IF NOT Execute THEN
	eState := STATE_RESETTING;
ELSIF _Error THEN
	eState := STATE_ERROR;
ELSIF _Abort THEN
	eState := STATE_ABORTING;
ELSIF _Executed THEN
	eState := STATE_DONE;
END_IF
END_METHOD

METHOD  M_STATE_RESETTING
VAR_INPUT
END_VAR
Busy := FALSE;
Aborted := FALSE;
Error := FALSE;

CASE uiResettingStep OF
	0:
		ModeRequestValid := FALSE;
		TON_WaitModeSwitch.IN := FALSE;

		uiResettingStep := 100;

	100:
		_ResetCompleted := TRUE;
END_CASE

IF _ResetCompleted THEN
	eState := STATE_DORMANT;
END_IF
END_METHOD

END_FUNCTION_BLOCK

// ---- Library/30_Simulation/10_IOSim/FB_SimulatedIO.TcPOU
(*
    FB_SimulatedIO — 數位孿生 IO 模擬層
    =====================================================
    每個 PLC 週期：
      1. 將所有安全門、氣壓 Input bit 強制為 TRUE（使機器可啟動）
      2. 監看 GVL_Output.uniDO.stDO 的 Valve 輸出位元
      3. 透過 TON 延遲後，回寫對應的 GVL_Input.uniDI.stDI 感測器位元
    使用方式：在 FB_MachineControl 主體中：
      IF EnableSimulation THEN fbSimulatedIO(); END_IF
*)
FUNCTION_BLOCK FB_SimulatedIO
VAR_INPUT
END_VAR
VAR_OUTPUT
END_VAR
VAR
    // ----- 安全輸入注入用旗標 -----
    _tSafetyInject : TON; // 短延遲確保每次都會執行注入

    // ----- Group 1: Double valve, FrontSensor + RearSensor -----
    // fbUpCV_DiameterHoriz
    tonDiamHoriz_Ext : TON;
    tonDiamHoriz_Ret : TON;
    // fbTransmitCV_CamaraHoriz
    tonCamaraHoriz_Ext : TON;
    tonCamaraHoriz_Ret : TON;

    // ----- Group 2: Single valve, FrontSensor + RearSensor -----
    // fbUpCV_DiameterVert
    tonDiamVert_Ext : TON;
    tonDiamVert_Ret : TON;
    // fbStackPush
    tonStackPush_Ext : TON;
    tonStackPush_Ret : TON;
    // fbAllocateRobot_LeftVert1
    tonLV1_Ext : TON;
    tonLV1_Ret : TON;
    // fbAllocateRobot_LeftVert2
    tonLV2_Ext : TON;
    tonLV2_Ret : TON;
    // fbAllocateRobot_RightVert1
    tonRV1_Ext : TON;
    tonRV1_Ret : TON;
    // fbAllocateRobot_RightVert2
    tonRV2_Ext : TON;
    tonRV2_Ret : TON;
    // fbRoundBelt_WorkZone_Plug
    tonWZPlug_Ext : TON;
    tonWZPlug_Ret : TON;
    // fbRoundBelt_ChargeZone_Plug
    tonCZPlug_Ext : TON;
    tonCZPlug_Ret : TON;
    // fbRoundBelt_TransmitCVZone_Plug
    tonTCVPlug_Ext : TON;
    tonTCVPlug_Ret : TON;
    // fbOutRobot_AsideVert
    tonAsideVert_Ext : TON;
    tonAsideVert_Ret : TON;
    // fbOutRobot_BsideVert
    tonBsideVert_Ext : TON;
    tonBsideVert_Ret : TON;

    // ----- Group 3: Double valve, RearSensor only -----
    // fbUpCV_Block1/2/3
    tonUpBlock1_Ext : TON;
    tonUpBlock1_Ret : TON;
    tonUpBlock2_Ext : TON;
    tonUpBlock2_Ret : TON;
    tonUpBlock3_Ext : TON;
    tonUpBlock3_Ret : TON;
    // fbLowCV_Block1/2
    tonLowBlock1_Ext : TON;
    tonLowBlock1_Ret : TON;
    tonLowBlock2_Ext : TON;
    tonLowBlock2_Ret : TON;
    // fbOutRobot_AsideClamp / BsideClamp
    tonAsideClamp_Ext : TON;
    tonAsideClamp_Ret : TON;
    tonBsideClamp_Ext : TON;
    tonBsideClamp_Ret : TON;

    // ----- Group 4: Single valve, RearSensor only -----
    // fbPullOutCV_AsideBlock / BsideBlock
    tonPullAside_Ext : TON;
    tonPullAside_Ret : TON;
    tonPullBside_Ext : TON;
    tonPullBside_Ret : TON;
    // fbRoundBelt_WorkZone_Press
    tonWZPress_Ext : TON;
    tonWZPress_Ret : TON;
    // fbDifferentSizeCV_Block1
    tonDiffBlock1_Ext : TON;
    tonDiffBlock1_Ret : TON;
    // fbSameSizeCV_Block1 / Block2
    tonSameBlock1_Ext : TON;
    tonSameBlock1_Ret : TON;
    tonSameBlock2_Ext : TON;
    tonSameBlock2_Ret : TON;
    // fbTurntable_Press
    tonTTPress_Ext : TON;
    tonTTPress_Ret : TON;
END_VAR
VAR CONSTANT
    tCYL_DELAY : TIME := T#300MS; // 汽缸模擬動作延遲（可依需求調整）
END_VAR

// ═══════════════════════════════════════════════════════════════
// 1. 安全輸入每週期強制 TRUE — 讓機器可以在無硬體下啟動
// ═══════════════════════════════════════════════════════════════
GVL_Input.uniDI.stDI.bSafetyDoor1  := TRUE;
GVL_Input.uniDI.stDI.bSafetyDoor2  := TRUE;
GVL_Input.uniDI.stDI.bSafetyDoor3  := TRUE;
GVL_Input.uniDI.stDI.bSafetyDoor4  := TRUE;
GVL_Input.uniDI.stDI.bSafetyDoor5  := TRUE;
GVL_Input.uniDI.stDI.bSafetyDoor6  := TRUE;
GVL_Input.uniDI.stDI.bSafetyDoor7  := TRUE;
GVL_Input.uniDI.stDI.bSafetyDoor8  := TRUE;
GVL_Input.uniDI.stDI.bSafetyDoor9  := TRUE;
GVL_Input.uniDI.stDI.bSafetyDoor10 := TRUE;
GVL_Input.uniDI.stDI.bSafetyDoor11 := TRUE;
GVL_Input.uniDI.stDI.bSafetyDoor12 := TRUE;
GVL_Input.uniDI.stDI.bSafetyDoor13 := TRUE;
GVL_Input.uniDI.stDI.bSafetyDoor14 := TRUE;
GVL_Input.uniDI.stDI.bAllocate_Electrical_Cabinet_SafetyDoor      := TRUE;
GVL_Input.uniDI.stDI.bShippingRobot_ElectricalCabinet_SafetyDoor  := TRUE;
GVL_Input.uniDI.stDI.bStorage_AirPressure_Ready   := TRUE;
GVL_Input.uniDI.stDI.bAllocate_AirPressure_Ready  := TRUE;

// ═══════════════════════════════════════════════════════════════
// 2. 汽缸 IO 模擬  (讀 Output Valve → 延遲 → 寫 Input Sensor)
//    每個 TON:  _Ext 監看伸出命令, _Ret 監看縮回命令
// ═══════════════════════════════════════════════════════════════

// ─── Group 1: Double valve, FrontSensor + RearSensor ─────────

// fbUpCV_DiameterHoriz (雙閥, 兩端感測器)
tonDiamHoriz_Ext(IN := GVL_Output.uniDO.stDO.bUpCV_DiameterHoriz_Extend_Valve, PT := tCYL_DELAY);
tonDiamHoriz_Ret(IN := GVL_Output.uniDO.stDO.bUpCV_DiameterHoriz_Retract_Valve, PT := tCYL_DELAY);
IF tonDiamHoriz_Ext.Q THEN
    GVL_Input.uniDI.stDI.bUpCV_DiameterHoriz_FrontSensor := TRUE;
    GVL_Input.uniDI.stDI.bUpCV_DiameterHoriz_RearSensor  := FALSE;
ELSIF tonDiamHoriz_Ret.Q THEN
    GVL_Input.uniDI.stDI.bUpCV_DiameterHoriz_FrontSensor := FALSE;
    GVL_Input.uniDI.stDI.bUpCV_DiameterHoriz_RearSensor  := TRUE;
END_IF

// fbTransmitCV_CamaraHoriz (雙閥, 兩端感測器)
tonCamaraHoriz_Ext(IN := GVL_Output.uniDO.stDO.bTransmitCV_CamaraHorizDifferentSide_Valve, PT := tCYL_DELAY);
tonCamaraHoriz_Ret(IN := GVL_Output.uniDO.stDO.bTransmitCV_CamaraHorizSameSizeSide_Valve,  PT := tCYL_DELAY);
IF tonCamaraHoriz_Ext.Q THEN
    GVL_Input.uniDI.stDI.bTransmit_CamaraHorizDifferentSizeSide_Sensor := TRUE;
    GVL_Input.uniDI.stDI.bTransmit_CamaraHorizSameSizeSide_Sensor      := FALSE;
ELSIF tonCamaraHoriz_Ret.Q THEN
    GVL_Input.uniDI.stDI.bTransmit_CamaraHorizDifferentSizeSide_Sensor := FALSE;
    GVL_Input.uniDI.stDI.bTransmit_CamaraHorizSameSizeSide_Sensor      := TRUE;
END_IF

// ─── Group 2: Single valve, FrontSensor + RearSensor ─────────

// fbUpCV_DiameterVert
tonDiamVert_Ext(IN :=      GVL_Output.uniDO.stDO.bUpCV_DiameterVert_Valve, PT := tCYL_DELAY);
tonDiamVert_Ret(IN := NOT  GVL_Output.uniDO.stDO.bUpCV_DiameterVert_Valve, PT := tCYL_DELAY);
IF tonDiamVert_Ext.Q THEN
    GVL_Input.uniDI.stDI.bUpCV_DiameterVert_FrontSensor := TRUE;
    GVL_Input.uniDI.stDI.bUpCV_DiameterVert_RearSensor  := FALSE;
ELSIF tonDiamVert_Ret.Q THEN
    GVL_Input.uniDI.stDI.bUpCV_DiameterVert_FrontSensor := FALSE;
    GVL_Input.uniDI.stDI.bUpCV_DiameterVert_RearSensor  := TRUE;
END_IF

// fbStackPush
tonStackPush_Ext(IN :=      GVL_Output.uniDO.stDO.bStackPush_Valve, PT := tCYL_DELAY);
tonStackPush_Ret(IN := NOT  GVL_Output.uniDO.stDO.bStackPush_Valve, PT := tCYL_DELAY);
IF tonStackPush_Ext.Q THEN
    GVL_Input.uniDI.stDI.bStackPush_Pusher_FrontSensor := TRUE;
    GVL_Input.uniDI.stDI.bStackPush_Pusher_RearSensor  := FALSE;
ELSIF tonStackPush_Ret.Q THEN
    GVL_Input.uniDI.stDI.bStackPush_Pusher_FrontSensor := FALSE;
    GVL_Input.uniDI.stDI.bStackPush_Pusher_RearSensor  := TRUE;
END_IF

// fbAllocateRobot_LeftVert1
tonLV1_Ext(IN :=      GVL_Output.uniDO.stDO.bAllocateRobot_LeftVert1_Valve, PT := tCYL_DELAY);
tonLV1_Ret(IN := NOT  GVL_Output.uniDO.stDO.bAllocateRobot_LeftVert1_Valve, PT := tCYL_DELAY);
IF tonLV1_Ext.Q THEN
    GVL_Input.uniDI.stDI.bAllocateRobot_LeftVert1_LowSensor  := TRUE;
    GVL_Input.uniDI.stDI.bAllocateRobot_LeftVert1_HighSensor := FALSE;
ELSIF tonLV1_Ret.Q THEN
    GVL_Input.uniDI.stDI.bAllocateRobot_LeftVert1_LowSensor  := FALSE;
    GVL_Input.uniDI.stDI.bAllocateRobot_LeftVert1_HighSensor := TRUE;
END_IF

// fbAllocateRobot_LeftVert2
tonLV2_Ext(IN :=      GVL_Output.uniDO.stDO.bAllocateRobot_LeftVert2_Valve, PT := tCYL_DELAY);
tonLV2_Ret(IN := NOT  GVL_Output.uniDO.stDO.bAllocateRobot_LeftVert2_Valve, PT := tCYL_DELAY);
IF tonLV2_Ext.Q THEN
    GVL_Input.uniDI.stDI.bAllocateRobot_LeftVert2_LowSensor  := TRUE;
    GVL_Input.uniDI.stDI.bAllocateRobot_LeftVert2_HighSensor := FALSE;
ELSIF tonLV2_Ret.Q THEN
    GVL_Input.uniDI.stDI.bAllocateRobot_LeftVert2_LowSensor  := FALSE;
    GVL_Input.uniDI.stDI.bAllocateRobot_LeftVert2_HighSensor := TRUE;
END_IF

// fbAllocateRobot_RightVert1
tonRV1_Ext(IN :=      GVL_Output.uniDO.stDO.bAllocateRobot_RightVert1_Valve, PT := tCYL_DELAY);
tonRV1_Ret(IN := NOT  GVL_Output.uniDO.stDO.bAllocateRobot_RightVert1_Valve, PT := tCYL_DELAY);
IF tonRV1_Ext.Q THEN
    GVL_Input.uniDI.stDI.bAllocateRobot_RightVert1_LowSensor  := TRUE;
    GVL_Input.uniDI.stDI.bAllocateRobot_RightVert1_HighSensor := FALSE;
ELSIF tonRV1_Ret.Q THEN
    GVL_Input.uniDI.stDI.bAllocateRobot_RightVert1_LowSensor  := FALSE;
    GVL_Input.uniDI.stDI.bAllocateRobot_RightVert1_HighSensor := TRUE;
END_IF

// fbAllocateRobot_RightVert2
tonRV2_Ext(IN :=      GVL_Output.uniDO.stDO.bAllocateRobot_RightVert2_Valve, PT := tCYL_DELAY);
tonRV2_Ret(IN := NOT  GVL_Output.uniDO.stDO.bAllocateRobot_RightVert2_Valve, PT := tCYL_DELAY);
IF tonRV2_Ext.Q THEN
    GVL_Input.uniDI.stDI.bAllocateRobot_RightVert2_LowSensor  := TRUE;
    GVL_Input.uniDI.stDI.bAllocateRobot_RightVert2_HighSensor := FALSE;
ELSIF tonRV2_Ret.Q THEN
    GVL_Input.uniDI.stDI.bAllocateRobot_RightVert2_LowSensor  := FALSE;
    GVL_Input.uniDI.stDI.bAllocateRobot_RightVert2_HighSensor := TRUE;
END_IF

// fbRoundBelt_WorkZone_Plug
tonWZPlug_Ext(IN :=      GVL_Output.uniDO.stDO.bRoundBelt_WorkZone_Plug_Valve, PT := tCYL_DELAY);
tonWZPlug_Ret(IN := NOT  GVL_Output.uniDO.stDO.bRoundBelt_WorkZone_Plug_Valve, PT := tCYL_DELAY);
IF tonWZPlug_Ext.Q THEN
    GVL_Input.uniDI.stDI.bRoundBelt_WorkZonePlug_frontSensor := TRUE;
    GVL_Input.uniDI.stDI.bRoundBelt_WorkZonePlug_RearSensor  := FALSE;
ELSIF tonWZPlug_Ret.Q THEN
    GVL_Input.uniDI.stDI.bRoundBelt_WorkZonePlug_frontSensor := FALSE;
    GVL_Input.uniDI.stDI.bRoundBelt_WorkZonePlug_RearSensor  := TRUE;
END_IF

// fbRoundBelt_ChargeZone_Plug
tonCZPlug_Ext(IN :=      GVL_Output.uniDO.stDO.bRoundBelt_ChargeZone_Plug_Valve, PT := tCYL_DELAY);
tonCZPlug_Ret(IN := NOT  GVL_Output.uniDO.stDO.bRoundBelt_ChargeZone_Plug_Valve, PT := tCYL_DELAY);
IF tonCZPlug_Ext.Q THEN
    GVL_Input.uniDI.stDI.bRoundBelt_ChangeZonePlug_FrontSensor := TRUE;
    GVL_Input.uniDI.stDI.bRoundBelt_ChangeZonePlug_RearSensor  := FALSE;
ELSIF tonCZPlug_Ret.Q THEN
    GVL_Input.uniDI.stDI.bRoundBelt_ChangeZonePlug_FrontSensor := FALSE;
    GVL_Input.uniDI.stDI.bRoundBelt_ChangeZonePlug_RearSensor  := TRUE;
END_IF

// fbRoundBelt_TransmitCVZone_Plug
tonTCVPlug_Ext(IN :=      GVL_Output.uniDO.stDO.bRoundBelt_TransmitCVZone_Plug_Valve, PT := tCYL_DELAY);
tonTCVPlug_Ret(IN := NOT  GVL_Output.uniDO.stDO.bRoundBelt_TransmitCVZone_Plug_Valve, PT := tCYL_DELAY);
IF tonTCVPlug_Ext.Q THEN
    GVL_Input.uniDI.stDI.bRoundBelt_TransmitCVZonePlug_FrontSensor := TRUE;
    GVL_Input.uniDI.stDI.bRoundBelt_TransmitCVZonePlug_RearSensor  := FALSE;
ELSIF tonTCVPlug_Ret.Q THEN
    GVL_Input.uniDI.stDI.bRoundBelt_TransmitCVZonePlug_FrontSensor := FALSE;
    GVL_Input.uniDI.stDI.bRoundBelt_TransmitCVZonePlug_RearSensor  := TRUE;
END_IF

// fbOutRobot_AsideVert (FrontSensor=Low, RearSensor=High)
tonAsideVert_Ext(IN :=      GVL_Output.uniDO.stDO.bOutRobot_AsideVert_Valve, PT := tCYL_DELAY);
tonAsideVert_Ret(IN := NOT  GVL_Output.uniDO.stDO.bOutRobot_AsideVert_Valve, PT := tCYL_DELAY);
IF tonAsideVert_Ext.Q THEN
    GVL_Input.uniDI.stDI.bOutRobot_AsideVert_LowSensor  := TRUE;
    GVL_Input.uniDI.stDI.bOutRobot_AsideVert_HighSensor := FALSE;
ELSIF tonAsideVert_Ret.Q THEN
    GVL_Input.uniDI.stDI.bOutRobot_AsideVert_LowSensor  := FALSE;
    GVL_Input.uniDI.stDI.bOutRobot_AsideVert_HighSensor := TRUE;
END_IF

// fbOutRobot_BsideVert (FrontSensor=Low, RearSensor=High)
tonBsideVert_Ext(IN :=      GVL_Output.uniDO.stDO.bOutRobot_BsideVert_Valve, PT := tCYL_DELAY);
tonBsideVert_Ret(IN := NOT  GVL_Output.uniDO.stDO.bOutRobot_BsideVert_Valve, PT := tCYL_DELAY);
IF tonBsideVert_Ext.Q THEN
    GVL_Input.uniDI.stDI.bOutRobot_BsideVert_LowSensor  := TRUE;
    GVL_Input.uniDI.stDI.bOutRobot_BsideVert_HighSensor := FALSE;
ELSIF tonBsideVert_Ret.Q THEN
    GVL_Input.uniDI.stDI.bOutRobot_BsideVert_LowSensor  := FALSE;
    GVL_Input.uniDI.stDI.bOutRobot_BsideVert_HighSensor := TRUE;
END_IF

// ─── Group 3: Double valve, RearSensor only ───────────────────

// fbUpCV_Block1  (Up=Extend=front, Down=Retract=rear)
tonUpBlock1_Ext(IN := GVL_Output.uniDO.stDO.bUpCV_Block1_Up_Valve,   PT := tCYL_DELAY);
tonUpBlock1_Ret(IN := GVL_Output.uniDO.stDO.bUpCV_Block1_Down_Valve, PT := tCYL_DELAY);
IF tonUpBlock1_Ext.Q THEN
    GVL_Input.uniDI.stDI.bUpCV_Block1_RearSensor := FALSE;
ELSIF tonUpBlock1_Ret.Q THEN
    GVL_Input.uniDI.stDI.bUpCV_Block1_RearSensor := TRUE;
END_IF

// fbUpCV_Block2
tonUpBlock2_Ext(IN := GVL_Output.uniDO.stDO.bUpCV_Block2_Up_Valve,   PT := tCYL_DELAY);
tonUpBlock2_Ret(IN := GVL_Output.uniDO.stDO.bUpCV_Block2_Down_Valve, PT := tCYL_DELAY);
IF tonUpBlock2_Ext.Q THEN
    GVL_Input.uniDI.stDI.bUpCV_Block2_RearSensor := FALSE;
ELSIF tonUpBlock2_Ret.Q THEN
    GVL_Input.uniDI.stDI.bUpCV_Block2_RearSensor := TRUE;
END_IF

// fbUpCV_Block3
tonUpBlock3_Ext(IN := GVL_Output.uniDO.stDO.bUpCV_Block3_Up_Valve,   PT := tCYL_DELAY);
tonUpBlock3_Ret(IN := GVL_Output.uniDO.stDO.bUpCV_Block3_Down_Valve, PT := tCYL_DELAY);
IF tonUpBlock3_Ext.Q THEN
    GVL_Input.uniDI.stDI.bUpCV_Block3_RearSensor := FALSE;
ELSIF tonUpBlock3_Ret.Q THEN
    GVL_Input.uniDI.stDI.bUpCV_Block3_RearSensor := TRUE;
END_IF

// fbLowCV_Block1  (Down=Extend, Up=Retract=rear)
tonLowBlock1_Ext(IN := GVL_Output.uniDO.stDO.bLowCV_Block1_Down_Valve, PT := tCYL_DELAY);
tonLowBlock1_Ret(IN := GVL_Output.uniDO.stDO.bLowCV_Block1_Up_Valve,   PT := tCYL_DELAY);
IF tonLowBlock1_Ext.Q THEN
    GVL_Input.uniDI.stDI.bLowCV_Block1_RearSensor := FALSE;
ELSIF tonLowBlock1_Ret.Q THEN
    GVL_Input.uniDI.stDI.bLowCV_Block1_RearSensor := TRUE;
END_IF

// fbLowCV_Block2
tonLowBlock2_Ext(IN := GVL_Output.uniDO.stDO.bLowCV_Block2_Down_Valve, PT := tCYL_DELAY);
tonLowBlock2_Ret(IN := GVL_Output.uniDO.stDO.bLowCV_Block2_Up_Valve,   PT := tCYL_DELAY);
IF tonLowBlock2_Ext.Q THEN
    GVL_Input.uniDI.stDI.bLowCV_Block2_RearSensor := FALSE;
ELSIF tonLowBlock2_Ret.Q THEN
    GVL_Input.uniDI.stDI.bLowCV_Block2_RearSensor := TRUE;
END_IF

// fbOutRobot_AsideClamp  (Close=Extend=front, Open=Retract=rear)
tonAsideClamp_Ext(IN := GVL_Output.uniDO.stDO.bOutRobot_AsideClamp_Close_Valve, PT := tCYL_DELAY);
tonAsideClamp_Ret(IN := GVL_Output.uniDO.stDO.bOutRobot_AsideClamp_Open_Valve,  PT := tCYL_DELAY);
IF tonAsideClamp_Ext.Q THEN
    GVL_Input.uniDI.stDI.bOutRobot_AsideClamp_RearSensor := FALSE;
ELSIF tonAsideClamp_Ret.Q THEN
    GVL_Input.uniDI.stDI.bOutRobot_AsideClamp_RearSensor := TRUE;
END_IF

// fbOutRobot_BsideClamp
tonBsideClamp_Ext(IN := GVL_Output.uniDO.stDO.bOutRobot_BsideClamp_Close_Valve, PT := tCYL_DELAY);
tonBsideClamp_Ret(IN := GVL_Output.uniDO.stDO.bOutRobot_BsideClamp_Open_Valve,  PT := tCYL_DELAY);
IF tonBsideClamp_Ext.Q THEN
    GVL_Input.uniDI.stDI.bOutRobot_BsideClamp_RearSensor := FALSE;
ELSIF tonBsideClamp_Ret.Q THEN
    GVL_Input.uniDI.stDI.bOutRobot_BsideClamp_RearSensor := TRUE;
END_IF

// ─── Group 4: Single valve, RearSensor only ───────────────────

// fbPullOutCV_AsideBlock
tonPullAside_Ext(IN :=      GVL_Output.uniDO.stDO.bPullOutCV_AsideBlock_Valve, PT := tCYL_DELAY);
tonPullAside_Ret(IN := NOT  GVL_Output.uniDO.stDO.bPullOutCV_AsideBlock_Valve, PT := tCYL_DELAY);
IF tonPullAside_Ext.Q THEN
    GVL_Input.uniDI.stDI.bPullOutCV_AsideBlock_RearSensor := FALSE;
ELSIF tonPullAside_Ret.Q THEN
    GVL_Input.uniDI.stDI.bPullOutCV_AsideBlock_RearSensor := TRUE;
END_IF

// fbPullOutCV_BsideBlock
tonPullBside_Ext(IN :=      GVL_Output.uniDO.stDO.bPullOutCV_BsideBlock_Valve, PT := tCYL_DELAY);
tonPullBside_Ret(IN := NOT  GVL_Output.uniDO.stDO.bPullOutCV_BsideBlock_Valve, PT := tCYL_DELAY);
IF tonPullBside_Ext.Q THEN
    GVL_Input.uniDI.stDI.bPullOutCV_BsideBlock_RearSensor := FALSE;
ELSIF tonPullBside_Ret.Q THEN
    GVL_Input.uniDI.stDI.bPullOutCV_BsideBlock_RearSensor := TRUE;
END_IF

// fbRoundBelt_WorkZone_Press (只有 RearSensor)
tonWZPress_Ext(IN :=      GVL_Output.uniDO.stDO.bRoundBelt_WorkZone_Press_Valve, PT := tCYL_DELAY);
tonWZPress_Ret(IN := NOT  GVL_Output.uniDO.stDO.bRoundBelt_WorkZone_Press_Valve, PT := tCYL_DELAY);
IF tonWZPress_Ext.Q THEN
    GVL_Input.uniDI.stDI.bRoundBelt_WorkZonePress_RearSensor := FALSE;
ELSIF tonWZPress_Ret.Q THEN
    GVL_Input.uniDI.stDI.bRoundBelt_WorkZonePress_RearSensor := TRUE;
END_IF

// fbDifferentSizeCV_Block1
tonDiffBlock1_Ext(IN :=      GVL_Output.uniDO.stDO.bDifferentSizeCV_Block1_Valve, PT := tCYL_DELAY);
tonDiffBlock1_Ret(IN := NOT  GVL_Output.uniDO.stDO.bDifferentSizeCV_Block1_Valve, PT := tCYL_DELAY);
IF tonDiffBlock1_Ext.Q THEN
    GVL_Input.uniDI.stDI.bDifferentCV_Block_RearSensor := FALSE;
ELSIF tonDiffBlock1_Ret.Q THEN
    GVL_Input.uniDI.stDI.bDifferentCV_Block_RearSensor := TRUE;
END_IF

// fbSameSizeCV_Block1
tonSameBlock1_Ext(IN :=      GVL_Output.uniDO.stDO.bSameSizeCV_Block1_Valve, PT := tCYL_DELAY);
tonSameBlock1_Ret(IN := NOT  GVL_Output.uniDO.stDO.bSameSizeCV_Block1_Valve, PT := tCYL_DELAY);
IF tonSameBlock1_Ext.Q THEN
    GVL_Input.uniDI.stDI.bSameSizeCVBlock1_RearSensor := FALSE;
ELSIF tonSameBlock1_Ret.Q THEN
    GVL_Input.uniDI.stDI.bSameSizeCVBlock1_RearSensor := TRUE;
END_IF

// fbSameSizeCV_Block2
tonSameBlock2_Ext(IN :=      GVL_Output.uniDO.stDO.bSameSizeCV_Block2_Valve, PT := tCYL_DELAY);
tonSameBlock2_Ret(IN := NOT  GVL_Output.uniDO.stDO.bSameSizeCV_Block2_Valve, PT := tCYL_DELAY);
IF tonSameBlock2_Ext.Q THEN
    GVL_Input.uniDI.stDI.bSameSizeCVBlock2_RearSensor := FALSE;
ELSIF tonSameBlock2_Ret.Q THEN
    GVL_Input.uniDI.stDI.bSameSizeCVBlock2_RearSensor := TRUE;
END_IF

// fbTurntable_Press (只有 RearSensor)
tonTTPress_Ext(IN :=      GVL_Output.uniDO.stDO.bTurntable_Press_Valve, PT := tCYL_DELAY);
tonTTPress_Ret(IN := NOT  GVL_Output.uniDO.stDO.bTurntable_Press_Valve, PT := tCYL_DELAY);
IF tonTTPress_Ext.Q THEN
    GVL_Input.uniDI.stDI.bTurnTable_Press_RearSensor := FALSE;
ELSIF tonTTPress_Ret.Q THEN
    GVL_Input.uniDI.stDI.bTurnTable_Press_RearSensor := TRUE;
END_IF

END_FUNCTION_BLOCK

// ---- Library/10_Machine/19_Device/FanucRobot/FB_FanucRobot_Basic.TcPOU
FUNCTION_BLOCK FB_FanucRobot_Basic IMPLEMENTS IBasicElement
VAR_INPUT
    Estop  : BOOL; // PLC ->send to Robot E-Stop
    OpMode : E_FanucRobotOpMode := RSR01; // Select Fanuc robot prog RSR1~RSR3
    Start  : BOOL;
    Reset  : BOOL; // Reset Fanuc Robot prog
    Hold   : BOOL; // PLC - > Robot send hold command
	ManualCtrl : REFERENCE TO ST_Manual_FanucRobot;
END_VAR

VAR_OUTPUT
    qEnable       : BOOL;
    qFault        : BOOL;
    E_Stop_Output : BOOL; // Touch pannel's E-Stop has been trig;
    Halt          : BOOL; // True : Robot in helt state.
    Error         : BOOL; // True : Robot has error
    ErrorID       : UDINT; // Error ID output
	ErrMsg 		  : T_MaxString;	  
END_VAR

VAR
    // Slot1
    _rawIn_UI AT %I*  : ARRAY[0..3] OF BYTE; // UI : Fanuc robot default input rawdate
    _rawOut_UO AT %Q* : ARRAY[0..3] OF BYTE; // UO : Fanuc robot default output rawdate
    // Slot2
    _rawIn_DI AT %I*           : ARRAY[0..31] OF BYTE; // DI : user define input rawdate
    _rawOut_DO AT %Q*          : ARRAY[0..31] OF BYTE; // DO : user define output rawdate
    _EIPConnectionState AT %I* : UINT; // EIP connection State (EL6652 to Fanuc Robot)
    _FanucEIPState AT %I*      : UINT; // EIP module links to FanucRobot state
    _UI1                       : ST_FanucUI1; // Fanuc Robot default Input
    _UO1                       : ST_FanucUO1; // Fanuc Robot default Output
    _DO1                       : ST_Fanuc_WarehouseHandshake; // Fanuc robot program's handshake for clampA warehouse pick / place box
    _DO2                       : ST_Fanuc_WarehouseHandshake; // Fanuc robot program's handshake for clampB warehouse pick / place box
    _DO3                       : ST_Fanuc_AbsMove; // Fanuc robot program's handshake for clampA to target area pick / place box
    _DO4                       : ST_Fanuc_AbsMove; // Fanuc robot program's handshake for clampB to target area pick / place box
    _DO5                       : ST_Fanuc_GeneralCommand; // Fanuc robot program's handshake for general control
    _DO6                       : ST_ReadWriteParaCmd; // Fanuc robot Read/Write parameter command 
    _DO7                       : INT; // Write process X position offset
    _DO8                       : INT; // Write process Y position offset
    _DO9                       : INT; // Write process Z position offset
    _DO10                      : INT; // Write process W position offset
    _DO11                      : INT; // Write process P position offset
    _DO12                      : INT; // Write process R position offset
    _Do13                      : INT; // Write process Area index
    _Do14                      : INT; // Write process Address index
    _Do15                      : INT; // Write process Layer index
    _DO16                      : INT; // Write process Slide index
    _DO17                      : ST_CCD_ZoneUse; // Set Robot use ccd or not.
    _DI1                       : ST_Fanuc_Status; // Fanuc robot program's handshake for process status
    _DI2                       : INT; // Readprocess X position offset
    _DI3                       : INT; // Read process Y position offset
    _DI4                       : INT; // Read process Z position offset
    _DI5                       : INT; // Read process W position offset
    _DI6                       : INT; // Read process P position offset
    _DI7                       : INT; // Read process R position offset
    _DI8                       : INT; // Read process Area index
    _DI9                       : INT; // Read process Address index
    _DI10                      : INT; // Read Process Layer index
    _DI11                      : INT; // Read Process Slide index
    _DI12                      : ST_ReadWriteParaStatus; // Read/Write process Status
    _VelocityCommand           : ST_IntToBool; // Robot coordenate velocity
    // Prog inside
    eState               : E_MethodStatus_Basic;
    uiRobotExecutingStep : UINT;
    uiRobotResettingStep : UINT;
    _Error               : BOOL;
    _Abort               : BOOL;
    TON_Restart_delay    : TON;
    TON_Reset_delay      : TON;
    Rtrig_RebootRobot    : R_TRIG;
    //fbReadSingleOffsetData  : FB_ReadSingleOffsetData;
    //fbWriteSingleOffsetData : FB_WriteSingleOffsetData;
    _Status               : T_MaxString;
    _eOpMode              : E_FanucRobotOpMode;
    _ModeChanging         : BOOL;
    _Completed            : BOOL;
    _ModeChanged          : BOOL;
    _uiRSR01_Step         : UINT;
    _uiRSR02_Step         : UINT;
    _uiRSR03_Step         : UINT;
    _RetryCount           : INT := 0;
    Ton_SetProgTimeOut    : TON; // This timer is used to counting the time to switch FanucRobot prog over range.
    _RSR1_Ready           : BOOL; // Fanuc Robot running in RSR1 prog, allow to Warehouse or AbsMove command.
    _RSR2_Completed       : BOOL; // Fanuc Robot finished the homing prog.
    _RSR3_Ready           : BOOL; // Fanuc Robot ready to work.
    TON_ResetFixDelay     : TON;
    Ton_RSR_SwitchDelay   : TON; // This timer is used to counting the time to switch rsr prog
    ErrorCode             : ST_IntToBool; // This value is which read from fanuc robot.
    Ton_START_SwitchDelay : TON; // This timer is used to counting the time to switch Start signal, Fanuc process need on 0.3s and off
END_VAR

VAR CONSTANT
    RetryMaxTimes   : INT  := 3;
    tSwitchProgTime : TIME := T#1S;
    tResetFixTime   : TIME := T#0.3S;
END_VAR

// Active base units.
A00_BaseUnit();
// Active mode controller
A10_ModeControl();
// Active state controller
A20_ErrorHandle();

Update();

ACTION A00_BaseUnit:
Ton_SetProgTimeOut(PT := tSwitchProgTime);
TON_Restart_delay(PT := T#1S); // Fanuc Robot need IMSTP on over 1s
TON_Reset_delay(PT := T#1S);
TON_ResetFixDelay(PT := tResetFixTime);
Ton_RSR_SwitchDelay(PT := T#0.3S);
Ton_START_SwitchDelay(PT := T#0.4S); // Fanuc Robot need on 0.3s and then set off
E_Stop_Output := _DI12.E_Stop;
END_ACTION

ACTION A10_ModeControl:
CASE _eOpMode OF
	E_FanucRobotOpMode.RSR01:
		M_ControlRSR01(bCompleted=> _Completed, ModeChanging=> _ModeChanging, ModeChanged=> _ModeChanged);
	E_FanucRobotOpMode.RSR02:
		M_ControlRSR02(bCompleted=> _Completed, ModeChanging=> _ModeChanging, ModeChanged=> _ModeChanged);
END_CASE
END_ACTION

ACTION A20_ErrorHandle:
ErrMsg := _Status;
END_ACTION

ACTION A20_StateControl:
TON_Restart_delay(PT := T#0.5S);
TON_Reset_delay(PT:=T#0.5S);
CASE eState OF
    E_MethodStatus_Basic.STATE_DORMANT:
        Enable(FALSE);
        M_Reset(FALSE);
        uiRobotExecutingStep := 0;
        uiRobotResettingStep := 0;

		IF _eOpMode = RSR01 OR _eOpMode = RSR02 OR _eOpMode = RSR03 THEN
			eState := E_MethodStatus_Basic.STATE_EXECUTING;
		END_IF
    E_MethodStatus_Basic.STATE_EXECUTING:
        CASE uiRobotExecutingStep OF
            0:
                Enable(iTrigger := TRUE);
                M_Reset(iTrigger := TRUE);
				TON_Reset_delay.in := TRUE;
                IF TON_Reset_delay.Q THEN
                    uiRobotExecutingStep := 100;
                END_IF
            100:
                M_Reset(iTrigger := FALSE);
				TON_Reset_delay.IN := FALSE;
                IF _UO1.UO01_CmdEnabled AND _UO1.UO02_SystemReady THEN
					_VelocityCommand.nInt := 1;
                    uiRobotExecutingStep := 200;
                END_IF
            200:
				// Clear Fanuc robot's action
				GVL_ADS.AutoMode_WarehouseMotoWithRobotMove.HandShake.Execute := FALSE;
				GVL_ADS.AutoMode_RobotAbsMove.HandShake.Execute := FALSE;
				_DO1.bExecute := FALSE; // Warehouse with robot clampA
				_DO2.bExecute := FALSE; // Warehouse with robot clampB
				_DO3.bExecute := FALSE; // AbsMove with robot clampA
				_DO4.bExecute := FALSE; // AbsMove with robot clampB
				uiRobotExecutingStep := 250;
			300:
				// Switch RSR3 and read all of offset data
				GVL_ADS.FanucRobot_ReadAllOffsetData.Command.Execute := TRUE;
				IF GVL_ADS.FanucRobot_ReadAllOffsetData.Status.Done THEN
					uiRobotExecutingStep := 400;
				ELSIF GVL_ADS.FanucRobot_ReadAllOffsetData.Status.Error THEN
					_Error := TRUE;
					_Status := 'FB_FanucRobot_Basic Step 300: Read All offset data failue';
				END_IF
			400:
                _UI1.UI09_RSR1 := TRUE;

                IF _UO1.UO11_ACK1 THEN
                    uiRobotExecutingStep := 500;
                END_IF
            500:
                _UI1.UI09_RSR1       := FALSE;
				_VelocityCommand.nInt := 30;
                uiRobotExecutingStep := 600;
            600: // Wait command
				_DO5.ClampA_Close :=  GVL_ADS.FanucRobot_General.Command.ClampA_Close;
				_DO5.ClampA_Open := GVL_ADS.FanucRobot_General.Command.ClampA_Open;
				_DO5.ClampB_Close := GVL_ADS.FanucRobot_General.Command.ClampB_Close;
				_DO5.ClampB_Open := GVL_ADS.FanucRobot_General.Command.ClampB_Open;
				_DO6.ByPassClampSensor := GVL_ADS.FanucRobot_General.Command.ByPassClampSensor;
				GVL_ADS.FanucRobot_General.Status.ClampA_Open := _DI1.ClampA_Open;
				GVL_ADS.FanucRobot_General.Status.ClampA_Sensor := _DI1.ClampA_Sensor;
				GVL_ADS.FanucRobot_General.Status.ClampB_Open := _DI1.ClampB_Open ;
				GVL_ADS.FanucRobot_General.Status.ClampB_Sensor := _DI1.ClampB_Sensor;
				_VelocityCommand.nInt := GVL_ADS.FanucRobot_General.Command.RobotVelocity;
        END_CASE

        IF (*qFault OR *)_Error THEN
            //Soft E-Stop will cause Fault error
            eState := E_MethodStatus_Basic.STATE_ERROR;
        ELSIF _Abort THEN
            eState := E_MethodStatus_Basic.STATE_ABORTING;
		ELSIF Estop THEN
			eState := E_MethodStatus_Basic.STATE_ABORTING;
        END_IF
    E_MethodStatus_Basic.STATE_DONE:
        ;
    E_MethodStatus_Basic.STATE_ABORTING:
	;
//        Hold();

        IF _UO1.UO04_PrgPaused THEN
            eState := E_MethodStatus_Basic.STATE_Aborted;
        END_IF
    E_MethodStatus_Basic.STATE_Aborted:
        IF _UI1.UI05_FaultReset OR GVL.Reset THEN
            eState := E_MethodStatus_Basic.STATE_RESETTING;
        END_IF
    E_MethodStatus_Basic.STATE_ERROR:
        IF _UI1.UI05_FaultReset THEN
            eState := E_MethodStatus_Basic.STATE_RESETTING;
        END_IF
    E_MethodStatus_Basic.STATE_RESETTING:
        CASE uiRobotResettingStep OF
            0:
                IF NOT _UO1.UO06_Fault THEN
                    IF NOT _UO1.UO04_PrgPaused THEN
                        uiRobotResettingStep := 1000;
                    ELSE
                        uiRobotResettingStep := 2000;
                    END_IF
                ELSE
                    uiRobotResettingStep := 1000;
                END_IF
            1000:
                M_Reset(TRUE);
				TON_Reset_delay.in := TRUE;
				IF TON_Reset_delay.Q THEN
                	uiRobotResettingStep := 1010;
				END_IF
            1010:
				TON_Reset_delay.IN :=FALSE;
                M_Reset(FALSE);
                uiRobotResettingStep := 9000;
            2000:
                _UI1.UI02_Hold       := TRUE;
                TON_Restart_delay.IN := TRUE; // TimeCount start

                IF TON_Restart_delay.Q THEN
                    uiRobotResettingStep := 2100;
                END_IF
            2100:
                TON_Restart_delay.IN := FALSE;
                _UI1.UI06_Start      := TRUE;
                uiRobotResettingStep := 9000;
            9000:
                IF NOT qFault THEN
                    eState := E_MethodStatus_Basic.STATE_DORMANT;
                END_IF
        END_CASE
END_CASE
Rtrig_RebootRobot(CLK:= GVL.MachineReset.AllReset);
IF Rtrig_RebootRobot.Q	AND qFault THEN
	ReBoot();
END_IF
END_ACTION

PROPERTY AbsMoveClampA_Handshake : ST_Fanuc_AbsMove
GET
AbsMoveClampA_Handshake := _DO3;
END_GET
SET
// Outside -> FB 
_DO3 := AbsMoveClampA_Handshake;
END_SET
END_PROPERTY

PROPERTY AbsMoveClampB_Handshake : ST_Fanuc_AbsMove
GET
AbsMoveClampB_Handshake := _DO4;
END_GET
SET
// Outside -> FB 
_DO4 := AbsMoveClampB_Handshake;
END_SET
END_PROPERTY

PROPERTY Bzone_AllowWork : Bool
GET
Bzone_AllowWork := THIS^._DO6.Bzone_AllowWork;
END_GET
SET
 THIS^._DO6.Bzone_AllowWork :=Bzone_AllowWork ;
END_SET
END_PROPERTY

PROPERTY BZoneInWork : Bool
GET
BZoneInWork := THIS^._DI12.BzoneInWork;
END_GET
END_PROPERTY

PROPERTY Command : ST_FanucUO1
GET
Command := _UO1;
END_GET
SET
_UO1 := Command;
END_SET
END_PROPERTY

METHOD Enable : BOOL
VAR_INPUT
iTrigger:BOOL;
END_VAR
VAR
	_RobotEnable:BOOL;
END_VAR
_RobotEnable:=iTrigger (*AND NOT Fault()*);

_UI1.UI01_IMSP:=_RobotEnable;
_UI1.UI02_Hold:=_RobotEnable;
_UI1.UI03_SFSP:=_RobotEnable;
_UI1.UI08_Enable:=_RobotEnable;
END_METHOD

METHOD EStop
VAR_INPUT
END_VAR
_UI1.UI03_SFSP:=FALSE;
END_METHOD

PROPERTY FanucRobot_MotionStatus : ST_Fanuc_Status
GET
FanucRobot_MotionStatus := _DI1;
END_GET
END_PROPERTY

METHOD Fault : BOOL
VAR_INPUT
END_VAR
VAR_INST
	bConectionError : BOOL;
END_VAR
bConectionError := (_EIPConnectionState <>0) OR (_FanucEIPState <> 0);
Fault:=_UO1.UO06_Fault OR _UO1.UO09_BattAlarm OR _DI1.Error OR bConectionError OR _UO1.UO08_TPEnabled;
END_METHOD

METHOD GetModelState
VAR_INPUT
END_VAR
VAR_OUTPUT
    xDone : BOOL;
    xBusy : BOOL;
    xError : BOOL;
    xAborted : BOOL;
    iErrorID : UDINT;
	UniqueErrorCode : STRING;
END_VAR
xError := Error;
iErrorID := INT_TO_UDINT(ErrorCode.nInt);
END_METHOD

METHOD GetName : STRING
VAR_INPUT
END_VAR
GetName := 'Fanuc Robot';
END_METHOD

METHOD Hold
VAR_INPUT
END_VAR
_UI1.UI02_Hold:=FALSE;
END_METHOD

PROPERTY Homed : Bool
GET
Homed := _RSR2_Completed OR _UO1.UO07_AtPerch;
END_GET
END_PROPERTY

PROPERTY LayerIndex : INT
SET
_Do15 := LayerIndex;
END_SET
END_PROPERTY

METHOD M_ActiveRSR01
VAR_INPUT
END_VAR
VAR_OUTPUT
	bCompleted : BOOL;
END_VAR
CASE eState OF
    E_MethodStatus_Basic.STATE_DORMANT:
        Enable(FALSE);
        M_Reset(FALSE);
        _uiRSR01_Step        := 0;
        uiRobotExecutingStep := 0;
        uiRobotResettingStep := 0;
        _RSR1_Ready          := FALSE;
        _RSR2_Completed      := FALSE;
        _RSR3_Ready          := FALSE;
        TON_Reset_delay.IN   := FALSE;
        _RSR1_Ready          := FALSE;

        IF _eOpMode = RSR01 OR _eOpMode = RSR02 OR _eOpMode = RSR03 THEN
            eState := E_MethodStatus_Basic.STATE_EXECUTING;
        END_IF
    E_MethodStatus_Basic.STATE_EXECUTING:
        CASE uiRobotExecutingStep OF
            0:
                Enable(iTrigger := TRUE);
                TON_Restart_delay.IN := TRUE;

                IF TON_Restart_delay.Q THEN
                    uiRobotExecutingStep := 10;
                END_IF
            10:
                TON_Restart_delay.IN := FALSE;
                M_Reset(iTrigger := TRUE);
                _UI1.UI04_CycleStop  := TRUE;
                TON_ResetFixDelay.IN := TRUE;

                IF TON_ResetFixDelay.Q THEN
                    uiRobotExecutingStep := 100;
                END_IF
            100:
                TON_ResetFixDelay.IN := FALSE;
                TON_Reset_delay.in   := TRUE;
                M_Reset(iTrigger := FALSE);
                _UI1.UI04_CycleStop := FALSE;

                IF TON_Reset_delay.Q THEN
                    IF _UO1.UO01_CmdEnabled AND _UO1.UO02_SystemReady THEN
                        _Error                := FALSE;
						Enable(iTrigger := TRUE); // 20250428 Albert
                        _VelocityCommand.nInt := 1;
                        uiRobotExecutingStep  := 200;
                    ELSIF Error THEN
                        eState := E_MethodStatus_Basic.STATE_ERROR;
                    END_IF
                END_IF
            200:
                // Clear Fanuc robot's action
                TON_Reset_delay.IN                                            := FALSE;
                GVL_ADS.AutoMode_WarehouseMotoWithRobotMove.HandShake.Execute := FALSE;
                GVL_ADS.AutoMode_RobotAbsMove.HandShake.Execute               := FALSE;
                _DO1.bExecute                                                 := FALSE; // Warehouse with robot clampA
                _DO2.bExecute                                                 := FALSE; // Warehouse with robot clampB
                _DO3.bExecute                                                 := FALSE; // AbsMove with robot clampA
                _DO4.bExecute                                                 := FALSE; // AbsMove with robot clampB
                uiRobotExecutingStep                                          := 300;
            300:
                // Active RSR1
                _UI1.UI09_RSR1         := TRUE;
                Ton_SetProgTimeOut.IN  := TRUE; // Switch to RSR1 start.
                Ton_RSR_SwitchDelay.IN := TRUE;

                IF _UO1.UO11_ACK1 THEN
                    uiRobotExecutingStep := 400;
                ELSIF Error OR Ton_SetProgTimeOut.Q THEN
                    _Error  := TRUE;
                    _Status := 'FB_FanucRobot_Basic Step 300: RSR1 has error when RSR1 active.';
                END_IF
            400:
                // Close RSR1 command
                Ton_SetProgTimeOut.IN := FALSE; // Switch to RSR1 close.

                IF Ton_RSR_SwitchDelay.Q THEN
                    _UI1.UI09_RSR1       := FALSE;
                    uiRobotExecutingStep := 500;
                END_IF
            500:
                // Allow Robot auto / manual job
                IF (GVL_ADS.AutoMode_RobotAbsMove.HandShake.Busy OR GVL_ADS.AutoMode_RobotAbsMove.HandShake.Done) AND
                    (GVL_ADS.AutoMode_WarehouseMotoWithRobotMove.HandShake.Busy OR GVL_ADS.AutoMode_WarehouseMotoWithRobotMove.HandShake.Done) (*AND
                    (GVL_ADS.ADS_MotoCalibrationData.WDataCore.HandShake.Busy OR GVL_ADS.ADS_MotoCalibrationData.WDataCore.HandShake.Done) AND
                    (GVL_ADS.ADS_MotoCalibrationData.AbslutCore.HandShake.Busy OR GVL_ADS.ADS_MotoCalibrationData.AbslutCore.HandShake.Done)*)
                    THEN
                    bCompleted := FALSE;
                ELSE
                    bCompleted := TRUE;
                END_IF
				_Status := 'FB_FanucRobot_Basic Step 500: Robot in Executing State';		//edit by min 20250913
				M_ManualService();
                //_VelocityCommand.nInt                           := GVL_ADS.FanucRobot_General.Command.RobotVelocity;
                _RSR1_Ready                                     := TRUE;

                IF _DI1.Error THEN
                    _Abort := TRUE;
                END_IF
        END_CASE

        IF _Abort THEN
            eState := E_MethodStatus_Basic.STATE_ABORTING;
        ELSIF Hold THEN
            eState := E_MethodStatus_Basic.STATE_Holding;
		ELSIF _UO1.UO06_Fault THEN
	        //_Abort := TRUE;

//			_Error  := TRUE;
//			_Status := 'Robot has fatal alarm';
//			eState  := E_MethodStatus_Basic.STATE_ERROR;
        END_IF
    E_MethodStatus_Basic.STATE_DONE:
        ;
    E_MethodStatus_Basic.STATE_ABORTING:
        eState := E_MethodStatus_Basic.STATE_ERROR;
    E_MethodStatus_Basic.STATE_Aborted:
        ;
    E_MethodStatus_Basic.STATE_ERROR:
        Enable(iTrigger := FALSE);
        _RSR1_Ready := FALSE;

        IF reset THEN
            eState := E_MethodStatus_Basic.STATE_RESETTING;
        END_IF

        IF NOT Estop AND NOT Error THEN
            eState := E_MethodStatus_Basic.STATE_RESETTING;
        END_IF
    E_MethodStatus_Basic.STATE_RESETTING:
		CASE uiRobotResettingStep OF
			0 : 
				_Error                   := FALSE;
				_Abort := false;
				_Status                  := '';
				M_ResetAllCommand();
				Ton_START_SwitchDelay.IN := FALSE;
				TON_Restart_delay.IN := FALSE;
				uiRobotResettingStep := 10;
			10:
				M_Reset(iTrigger :=TRUE);
				TON_Restart_delay.IN := TRUE;
				IF TON_Restart_delay.Q THEN
					M_EnableWith4Input(TRUE	,TRUE,TRUE,FALSE);
					uiRobotResettingStep := 20;
				END_IF
			20:
				TON_Restart_delay.IN := FALSE;
				M_Reset(iTrigger :=FALSE);
        		//Enable(iTrigger := TRUE);
				IF NOT  _UO1.UO06_Fault THEN
					M_EnableWith4Input(TRUE	,TRUE,TRUE,FALSE);
					uiRobotResettingStep := 50;
				END_IF
				IF reset THEN
					uiRobotResettingStep := 0;
				END_IF
			30 :
				M_Reset(iTrigger :=TRUE);
				uiRobotResettingStep := 40;
			40:
				M_Reset(iTrigger :=FALSE);
				uiRobotResettingStep := 50;
			50:
				IF reset THEN
					uiRobotResettingStep := 0;
				END_IF
				IF NOT Error THEN
					eState := E_MethodStatus_Basic.STATE_DORMANT;
				END_IF
		END_CASE
    E_MethodStatus_Basic.STATE_Holding:
        _UI1.UI02_Hold := FALSE;

        IF _UO1.UO04_PrgPaused AND NOT _UO1.UO03_PrgRunning THEN
            Halt    := TRUE;
            _Status := 'FB_FanucRobot_Basic: Robot in Halt State';
            eState  := E_MethodStatus_Basic.STATE_Held;
        END_IF
		IF reset THEN
			eState         := E_MethodStatus_Basic.STATE_ERROR;
		END_IF
    E_MethodStatus_Basic.STATE_Held:
		Ton_START_SwitchDelay.IN := FALSE;
        IF reset AND NOT Hold THEN
			//M_Reset(iTrigger:=TRUE);		//edit by min , if need resume robot motion dont set robot UI04 cyclestop
			_UI1.UI05_FaultReset:=TRUE;
            Halt := FALSE;
		ELSE
			M_Reset(iTrigger :=FALSE);
        END_IF

        IF NOT Halt AND Start THEN
            _UI1.UI02_Hold := TRUE;
            eState         := E_MethodStatus_Basic.STATE_UnHold;
        END_IF
    E_MethodStatus_Basic.STATE_UnHold:
        Ton_START_SwitchDelay.IN := TRUE;
		 _UI1.UI09_RSR1         := TRUE;
        _UI1.UI06_Start          := NOT Ton_START_SwitchDelay.Q;
		
        IF NOT _UO1.UO04_PrgPaused AND _UO1.UO03_PrgRunning AND NOT _UI1.UI06_Start THEN
            Ton_START_SwitchDelay.IN := FALSE;
			 _UI1.UI09_RSR1         := FALSE;
            eState                   := E_MethodStatus_Basic.STATE_EXECUTING;
        END_IF
END_CASE

IF Estop THEN
   // _Error  := TRUE;
    _Status := 'FB_FanucRobot_Basic: EStop has been trigged.';
	eState  := E_MethodStatus_Basic.STATE_ERROR;
ELSIF _UO1.UO08_TPEnabled THEN
    _Error  := TRUE;
    _Status := 'FB_FanucRobot_Basic: TP has got contol';
	eState  := E_MethodStatus_Basic.STATE_ERROR;
ELSIF _UO1.UO09_BattAlarm THEN
    _Error  := TRUE;
    _Status := 'FB_FanucRobot_Basic: Robot has Battary alarm';
	eState  := E_MethodStatus_Basic.STATE_ERROR;
END_IF
END_METHOD

METHOD M_ActiveRSR02
VAR_INPUT
END_VAR
VAR_OUTPUT
	bCompleted : BOOL;
END_VAR
CASE eState OF
	E_MethodStatus_Basic.STATE_DORMANT:
        Enable(FALSE);
        M_Reset(FALSE);
        _uiRSR01_Step := 0;
		uiRobotExecutingStep := 0;
        uiRobotResettingStep := 0;
		_RSR1_Ready := FALSE;
		_RSR2_Completed := FALSE;
		_RSR3_Ready:=FALSE;
		TON_Reset_delay.IN := FALSE;
		IF _eOpMode = RSR01 OR _eOpMode = RSR02 OR _eOpMode = RSR03 THEN
			eState := E_MethodStatus_Basic.STATE_EXECUTING;
		END_IF
	E_MethodStatus_Basic.STATE_EXECUTING:
		CASE uiRobotExecutingStep OF
			0:
                Enable(iTrigger := TRUE);
				TON_Restart_delay.IN := TRUE;
				IF TON_Restart_delay.Q THEN
					uiRobotExecutingStep := 10;
				END_IF
			10:
				TON_Restart_delay.IN := FALSE;
                M_Reset(iTrigger := TRUE);
				TON_ResetFixDelay.in := TRUE;
				_UI1.UI04_CycleStop := TRUE;
				IF TON_ResetFixDelay.Q THEN
	                uiRobotExecutingStep := 100;
				END_IF
			100:
				TON_ResetFixDelay.in := FALSE;
				TON_Reset_delay.in := TRUE;
                M_Reset(iTrigger := FALSE);
				_UI1.UI04_CycleStop := FALSE;
				IF TON_Reset_delay.Q THEN
					IF _UO1.UO01_CmdEnabled AND _UO1.UO02_SystemReady THEN
						_VelocityCommand.nInt := 1;
						uiRobotExecutingStep := 200;
					ELSIF Error THEN
						eState := E_MethodStatus_Basic.STATE_ERROR;
					END_IF
				END_IF
			200:
				// Clear Fanuc robot's action
				GVL_ADS.AutoMode_WarehouseMotoWithRobotMove.HandShake.Execute := FALSE;
				GVL_ADS.AutoMode_RobotAbsMove.HandShake.Execute := FALSE;
				_DO1.bExecute := FALSE;
				_DO2.bExecute := FALSE;
				_DO3.bExecute := FALSE;
				_DO4.bExecute := FALSE;
				uiRobotExecutingStep := 300;
			300:
				// Switch RSR02
				_UI1.UI10_RSR2 := TRUE;
		
				IF _UO1.UO12_ACK2 THEN
					uiRobotExecutingStep := 400;
				END_IF
			400:
				_UI1.UI10_RSR2 := FALSE;
				IF (_DI1.Done OR _UO1.UO07_AtPerch )  
				THEN
					uiRobotExecutingStep := 9900;
				END_IF
			9900:
				eState := E_MethodStatus_Basic.STATE_DONE;
		END_CASE
	E_MethodStatus_Basic.STATE_DONE:
		_RSR2_Completed := TRUE;
		bCompleted := TRUE;
	E_MethodStatus_Basic.STATE_ABORTING:
		;
	E_MethodStatus_Basic.STATE_Aborted:
		;
	E_MethodStatus_Basic.STATE_ERROR:
		Enable(iTrigger := FALSE);
		IF reset THEN
			eState := E_MethodStatus_Basic.STATE_RESETTING;
		END_IF
		IF NOT Estop AND NOT Error THEN
			eState := E_MethodStatus_Basic.STATE_RESETTING;
		END_IF
	E_MethodStatus_Basic.STATE_RESETTING:
		eState := E_MethodStatus_Basic.STATE_DORMANT;
END_CASE
IF Estop OR _UO1.UO08_TPEnabled THEN
	eState := E_MethodStatus_Basic.STATE_ERROR;
	_Error := TRUE;
	_Status := 'FB_FanucRobot_Basic: EStop has been trigged.';
END_IF
END_METHOD

METHOD M_ActiveRSR03
VAR_INPUT
END_VAR
VAR_OUTPUT
	bCompleted : BOOL;
END_VAR
CASE _uiRSR03_Step OF
	0:
		// Stop Prog
		_RSR1_Ready := FALSE;
		_RSR2_Completed := FALSE;
		_RSR3_Ready:=FALSE;
		_UI1.UI04_CycleStop := TRUE;
		IF NOT _UO1.UO04_PrgPaused AND NOT _UO1.UO03_PrgRunning THEN
			_uiRSR03_Step := 100;
		END_IF
	100:
		// Close cycle stop
		_UI1.UI04_CycleStop := FALSE;
		// Set current prog - RSR03
		_UI1.UI11_RSR3 := TRUE;
		IF _UO1.UO13_ACK3 THEN
			_uiRSR03_Step := 200;
		END_IF
	200:
		// Clear RSR03 command 
		_UI1.UI11_RSR3 := FALSE;
		_uiRSR03_Step := 300;
	300:
		// Allow Read / Write offset data
		IF ( GVL_ADS.FanucRobot_ReadAllOffsetData.Status.Busy  OR GVL_ADS.FanucRobot_ReadAllOffsetData.Status.Done) AND
			(GVL_ADS.FanucRobot_ReadSingleOffsetData.Status.Busy OR GVL_ADS.FanucRobot_ReadSingleOffsetData.Status.Done) AND
			(GVL_ADS.FanucRobot_WirteSingleOffsetData.Status.Busy OR GVL_ADS.FanucRobot_WirteSingleOffsetData.Status.Done ) AND
			(GVL_ADS.FanucRobot_WriteAllOffsetData.Status.Busy OR GVL_ADS.FanucRobot_WriteAllOffsetData.Status.Done) 
		THEN
			_RSR3_Ready := FALSE;
			bCompleted := FALSE;
		ELSE
			_RSR3_Ready := FALSE;
			bCompleted := TRUE;
		END_IF 
		
END_CASE

CASE eState OF
	E_MethodStatus_Basic.STATE_DORMANT:
        Enable(FALSE);
        M_Reset(FALSE);
        _uiRSR01_Step := 0;
		uiRobotExecutingStep := 0;
        uiRobotResettingStep := 0;
		_RSR1_Ready := FALSE;
		_RSR2_Completed := FALSE;
		_RSR3_Ready:=FALSE;
		TON_Reset_delay.IN := FALSE;
		IF _eOpMode = RSR01 OR _eOpMode = RSR02 OR _eOpMode = RSR03 THEN
			eState := E_MethodStatus_Basic.STATE_EXECUTING;
		END_IF
	E_MethodStatus_Basic.STATE_EXECUTING:
		CASE uiRobotExecutingStep OF
			0:
                Enable(iTrigger := TRUE);
				TON_Restart_delay.IN := TRUE;
				IF TON_Restart_delay.Q THEN
					uiRobotExecutingStep := 10;
				END_IF
			10:
				TON_Restart_delay.IN := FALSE;
                M_Reset(iTrigger := TRUE);
				_UI1.UI04_CycleStop := TRUE;
				TON_ResetFixDelay.IN := TRUE;
				IF TON_ResetFixDelay.Q THEN
                	uiRobotExecutingStep := 100;
				END_IF
			100:
				TON_ResetFixDelay.IN := FALSE;
				TON_Reset_delay.in := TRUE;
                M_Reset(iTrigger := FALSE);
				_UI1.UI04_CycleStop := FALSE;
				IF TON_Reset_delay.Q THEN
					IF _UO1.UO01_CmdEnabled AND _UO1.UO02_SystemReady THEN
						_VelocityCommand.nInt := 1;
						uiRobotExecutingStep := 200;
					ELSIF Error THEN
						eState := E_MethodStatus_Basic.STATE_ERROR;
					END_IF
				END_IF
			200:
				// Clear Fanuc robot's action
				TON_Reset_delay.IN := FALSE;
				GVL_ADS.AutoMode_WarehouseMotoWithRobotMove.HandShake.Execute := FALSE;
				GVL_ADS.AutoMode_RobotAbsMove.HandShake.Execute := FALSE;
				_DO1.bExecute := FALSE; // Warehouse with robot clampA
				_DO2.bExecute := FALSE; // Warehouse with robot clampB
				_DO3.bExecute := FALSE; // AbsMove with robot clampA
				_DO4.bExecute := FALSE; // AbsMove with robot clampB
				uiRobotExecutingStep := 300;
			300:
				// Active RSR1
                _UI1.UI11_RSR3 := TRUE;
                IF _UO1.UO13_ACK3 THEN
                    uiRobotExecutingStep := 400;
				ELSIF Error THEN
					_Error := TRUE;
					_Status:='FB_FanucRobot_Basic Step 300: RSR3 has error when RSR3 active.';
                END_IF
			400:
				// Allow Read / Write offset data
				IF ( GVL_ADS.FanucRobot_ReadAllOffsetData.Status.Busy  OR GVL_ADS.FanucRobot_ReadAllOffsetData.Status.Done) AND
					(GVL_ADS.FanucRobot_ReadSingleOffsetData.Status.Busy OR GVL_ADS.FanucRobot_ReadSingleOffsetData.Status.Done) AND
					(GVL_ADS.FanucRobot_WirteSingleOffsetData.Status.Busy OR GVL_ADS.FanucRobot_WirteSingleOffsetData.Status.Done ) AND
					(GVL_ADS.FanucRobot_WriteAllOffsetData.Status.Busy OR GVL_ADS.FanucRobot_WriteAllOffsetData.Status.Done) 
				THEN
					_RSR3_Ready := FALSE;
					bCompleted := FALSE;
				ELSE
					_RSR3_Ready := FALSE;
					bCompleted := TRUE;
				END_IF 
		END_CASE
	E_MethodStatus_Basic.STATE_DONE:
		;
	E_MethodStatus_Basic.STATE_ABORTING:
		;
	E_MethodStatus_Basic.STATE_Aborted:
		;
	E_MethodStatus_Basic.STATE_ERROR:
		Enable(iTrigger := FALSE);
		IF Reset THEN
			eState := E_MethodStatus_Basic.STATE_RESETTING;
		END_IF
		IF  Estop AND NOT Error THEN
			eState := E_MethodStatus_Basic.STATE_RESETTING;
		END_IF
	E_MethodStatus_Basic.STATE_RESETTING:
		eState := E_MethodStatus_Basic.STATE_DORMANT;
END_CASE

IF Estop OR _UO1.UO08_TPEnabled THEN
	eState := E_MethodStatus_Basic.STATE_ERROR;
	_Error := TRUE;
	_Status := 'FB_FanucRobot_Basic: EStop has been trigged.';
END_IF
END_METHOD

METHOD M_ClearState : BOOL;
VAR_INPUT
END_VAR

eState := E_MethodStatus_Basic.STATE_DORMANT;
uiRobotExecutingStep := 0;
uiRobotResettingStep := 0;
M_ClearState := TRUE;
END_METHOD

METHOD M_ControlRSR01
VAR_INPUT
END_VAR
VAR_OUTPUT
	bCompleted : BOOL;
	ModeChanging : BOOL;
	ModeChanged : BOOL;
END_VAR
ModeChanging := FALSE;
ModeChanged := TRUE;
M_ActiveRSR01(bCompleted => bCompleted);

IF OpMode <> _eOpMode (*AND bCompleted*) THEN
    _uiRSR01_Step := 0;
    eState := E_MethodStatus_Basic.STATE_DORMANT;
    _eOpMode := OpMode;
END_IF
END_METHOD

METHOD M_ControlRSR02
VAR_INPUT
END_VAR
VAR_OUTPUT
    bCompleted : BOOL;
    ModeChanging : BOOL;
    ModeChanged : BOOL;
END_VAR
ModeChanging := FALSE;
ModeChanged := TRUE;
M_ActiveRSR02(bCompleted => bCompleted);

IF OpMode <> _eOpMode AND bCompleted THEN
    _uiRSR02_Step := 0;
    eState := E_MethodStatus_Basic.STATE_DORMANT;
    _eOpMode := OpMode;
END_IF
END_METHOD

METHOD M_ControlRSR03

VAR_INPUT
END_VAR
VAR_OUTPUT
    bCompleted : BOOL;
    ModeChanging : BOOL;
    ModeChanged : BOOL;
END_VAR
ModeChanging := FALSE;
ModeChanged := TRUE;
M_ActiveRSR03(bCompleted => bCompleted);

IF OpMode <> _eOpMode AND bCompleted THEN
	_uiRSR03_Step := 0;
	eState := E_MethodStatus_Basic.STATE_DORMANT;
	_eOpMode := OpMode;
END_IF
END_METHOD

METHOD PRIVATE M_EnableWith4Input : BOOL
VAR_INPUT
	IMSP : BOOL;
	Hold : BOOL;
	SFSP : BOOL;
	Enable : BOOL;
END_VAR
_UI1.UI01_IMSP:=IMSP;
_UI1.UI02_Hold:=Hold;
_UI1.UI03_SFSP:=SFSP;
_UI1.UI08_Enable:=Enable;
END_METHOD

METHOD M_GetErrorCode : Int
VAR_INPUT
END_VAR
ErrorCode.BitList.Bit0 := _DI1.ErrorID_01;
ErrorCode.BitList.Bit1 := _DI1.ErrorID_02;
ErrorCode.BitList.Bit2 := _DI1.ErrorID_03;
ErrorCode.BitList.Bit3 := _DI1.ErrorID_04;
ErrorCode.BitList.Bit4 := _DI1.ErrorID_05;
ErrorCode.BitList.Bit5 := _DI1.ErrorID_06;
ErrorCode.BitList.Bit6 := _DI1.ErrorID_07;
ErrorCode.BitList.Bit7 := _DI1.ErrorID_08;		
//ErrorCode.BitList.Bit8 := _DI1.ErrorID_09;
//ErrorCode.BitList.Bit9 := _DI1.ErrorID_10;
M_GetErrorCode := ErrorCode.nInt;
END_METHOD

METHOD M_Kawasaki_API
VAR_INPUT
	WarehouseClampA_Handshake : UINT;
	WarehouseClampB_Handshake : UINT;
	AbsMoveClampA_Handshake : UINT;
	AbsMoveClampB_Handshake : UINT;
END_VAR
VAR_OUTPUT
	Status : UINT;
END_VAR
MEMMOVE(destAddr:=ADR(_DO1),srcAddr:=ADR(WarehouseClampA_Handshake),n:=2);
MEMMOVE(destAddr:=ADR(_DO2),srcAddr:=ADR(WarehouseClampB_Handshake),n:=2);
MEMMOVE(destAddr:=ADR(_DO3),srcAddr:=ADR(AbsMoveClampA_Handshake),n:=2);
MEMMOVE(destAddr:=ADR(_DO4),srcAddr:=ADR(AbsMoveClampB_Handshake),n:=2);
IF NOT _UO1.UO08_TPEnabled THEN
	MEMMOVE(destAddr:=ADR(Status),srcAddr:=ADR(_DI1),n:=2);
END_IF
END_METHOD

METHOD M_ManualService
VAR_INPUT
END_VAR
_DO5.ClampA_Close := ManualCtrl.ClampA_Close;
_DO5.ClampA_Open := ManualCtrl.ClampA_Open;
_DO5.ClampB_Close := ManualCtrl.ClampB_Close;
_DO5.ClampB_Open := ManualCtrl.ClampB_Open;
_DO6.ByPassClampSensor := ManualCtrl.ByPassClampSensor;
GVL_ADS.FanucRobot_General.Status.ClampA_Open := _DI1.ClampA_Open;
GVL_ADS.FanucRobot_General.Status.ClampA_Sensor := _DI1.ClampA_Sensor;
GVL_ADS.FanucRobot_General.Status.ClampB_Open := _DI1.ClampB_Open;
GVL_ADS.FanucRobot_General.Status.ClampB_Sensor := _DI1.ClampB_Sensor;
END_METHOD

METHOD M_Reset : BOOL
VAR_INPUT
	iTrigger:BOOL;
END_VAR
_UI1.UI05_FaultReset:=iTrigger;
_UI1.UI04_CycleStop:=iTrigger;
END_METHOD

METHOD M_ResetAbsMoveClampACommand : BOOL
VAR_INPUT
END_VAR
VAR
	SpareData : ST_Fanuc_AbsMove;
END_VAR
_DO3 := SpareData;

M_ResetAbsMoveClampACommand := TRUE; // Method end
END_METHOD

METHOD M_ResetAbsMoveClampBCommand : BOOL
VAR_INPUT
END_VAR
VAR
	SpareData : ST_Fanuc_AbsMove;
END_VAR
_DO4 := SpareData;

M_ResetAbsMoveClampBCommand := true; // Method end
END_METHOD

METHOD M_ResetAbsMoveCommand : BOOL
VAR_INPUT
END_VAR
// Clear AbsMove ClampA command data
M_ResetAbsMoveClampACommand();
// Clear AbsMove ClampB command data
M_ResetAbsMoveClampBCommand();

M_ResetAbsMoveCommand := TRUE; // Method end
END_METHOD

METHOD M_ResetAllCommand : BOOL
VAR_INPUT
END_VAR
// Clear WareHouse command
M_ResetWareHouseCommand();
// Clear AbsMove Command
M_ResetAbsMoveCommand();

M_ResetAllCommand := TRUE; // Method end
END_METHOD

METHOD M_ResetMoveBoxToFeedInConveyor_ClampA : BOOL
VAR_INPUT
END_VAR
VAR
	SpaceData : ST_Fanuc_AbsMove;
END_VAR
_DO3 := SpaceData;

M_ResetMoveBoxToFeedInConveyor_ClampA := TRUE; // Mehtod end
END_METHOD

METHOD M_ResetMoveBoxToFeedInConveyor_ClampB : BOOL
VAR_INPUT
END_VAR
VAR
    SpaceData : ST_Fanuc_AbsMove;
END_VAR
_DO4 := SpaceData;

M_ResetMoveBoxToFeedInConveyor_ClampB := TRUE; // Method end
END_METHOD

METHOD M_ResetMoveBoxToFeedInConveyor_ClampBoth : BOOL
VAR_INPUT
END_VAR
VAR
    SpaceData : ST_Fanuc_AbsMove;
END_VAR
_DO3 := SpaceData;
_DO4 := SpaceData;

M_ResetMoveBoxToFeedInConveyor_ClampBoth := TRUE; // Method end
END_METHOD

METHOD M_ResetMoveBoxToRoundBelt_Both : BOOL
VAR_INPUT
END_VAR
VAR
    SpaceData : ST_Fanuc_AbsMove;
END_VAR
_DO3 := SpaceData;
_DO4 := SpaceData;

M_ResetMoveBoxToRoundBelt_Both := TRUE; // Method end
END_METHOD

METHOD M_ResetPullOutConveyorPickUpBox_ClampA : BOOL
VAR_INPUT
END_VAR
VAR
	SpaceData : ST_Fanuc_AbsMove;
END_VAR
_DO3 := SpaceData;

M_ResetPullOutConveyorPickUpBox_ClampA := TRUE; // Method end
END_METHOD

METHOD M_ResetPullOutConveyorPickUpBox_ClampB : BOOL
VAR_INPUT
END_VAR
VAR
    SpaceData : ST_Fanuc_AbsMove;
END_VAR
_DO4 := SpaceData;

M_ResetPullOutConveyorPickUpBox_ClampB := true; // Method end
END_METHOD

METHOD M_ResetPullOutConveyorPickUpBox_ClampBoth : BOOL
VAR_INPUT
END_VAR
VAR
    SpaceData : ST_Fanuc_AbsMove;
END_VAR
_DO3 := SpaceData;
_DO4 := SpaceData;

M_ResetPullOutConveyorPickUpBox_ClampBoth := TRUE; // Method end
END_METHOD

METHOD PUBLIC M_ResetRobotAbsMove : BOOL
VAR_INPUT
	ResetClampA : BOOL;
	ResetClampB : BOOL;
END_VAR

VAR
	SpaceData : ST_Fanuc_AbsMove;
END_VAR
IF ResetClampA THEN
	_DO3 := SpaceData;
END_IF

IF ResetClampB THEN
	_DO4 := SpaceData;
END_IF

M_ResetRobotAbsMove:=True;
END_METHOD

METHOD M_ResetWareHouseClampACommand : BOOL
VAR_INPUT
END_VAR
VAR
	SpareData : ST_Fanuc_WarehouseHandshake;
END_VAR
_DO1 := SpareData;

M_ResetWareHouseClampACommand := TRUE; // Method end
END_METHOD

METHOD M_ResetWareHouseClampBCommand : BOOL
VAR_INPUT
END_VAR
VAR
	SpareData : ST_Fanuc_WarehouseHandshake;
END_VAR
_DO2 := SpareData;

M_ResetWareHouseClampBCommand := true; // Method end
END_METHOD

METHOD M_ResetWareHouseCommand : BOOL
VAR_INPUT
END_VAR
// Clear WareHouse ClampA command data
M_ResetWareHouseClampACommand();
// Clear WareHouse ClampB command data
M_ResetWareHouseClampBCommand();

M_ResetWareHouseCommand := TRUE; // Method end
END_METHOD

METHOD M_ResetWareHousePickUpBox_ClampA : BOOL
VAR_INPUT
END_VAR
VAR
	SpaceData :ST_Fanuc_WarehouseHandshake;
END_VAR
// Clear command
_DO1 := SpaceData;

M_ResetWareHousePickUpBox_ClampA := TRUE; // Method End
END_METHOD

METHOD M_ResetWareHousePickUpBox_ClampB : BOOL
VAR_INPUT
END_VAR
VAR
	SpaceData :ST_Fanuc_WarehouseHandshake;
END_VAR
// Clear command
_DO2 := SpaceData;

M_ResetWareHousePickUpBox_ClampB := TRUE; // Method End
END_METHOD

METHOD M_ResetWareHousePickUpBox_ClampBoth : BOOL
VAR_INPUT
END_VAR
VAR
	SpaceData :ST_Fanuc_WarehouseHandshake;
END_VAR
// Clear command
_DO1 := SpaceData;
_DO2 := SpaceData;

M_ResetWareHousePickUpBox_ClampBoth := TRUE; // Method end
END_METHOD

(* This Method is used to send command data to Fanuc Robot, only clampA is work 
*)
METHOD M_StartAbsMoveAction_ClampA : BOOL
VAR_INPUT
	TargetArea : E_RobotArea; // Select the zone where robot will going.
	TargetAddress : E_RobotAddress; // Because the address num in different zone, the number define is different. But also need >= 1, 0 = undefined
	ClampAction : E_ClampAction; // need to define the command
	BoxReady : BOOL; // Fanuc robot prog will stop at a safe position just before reaching the target location, until `AllowContinue` is set to true.
END_VAR

VAR_OUTPUT
    Error  : BOOL;
    ErrMsg : T_MaxString;
END_VAR

VAR_INST
	_Area : ST_IntToBool;
	_Address : ST_IntToBool;
END_VAR
// Set target area
_Area.nInt := TargetArea;

CASE TargetArea OF
    E_RobotArea.RoundBelt..E_RobotArea.PullOutConveyor:
        _Area.nInt := TargetArea;
ELSE
    Error  := TRUE;
    ErrMsg := 'ClampA target area out of range';
	RETURN;
END_CASE

// Set target address
_Address.nInt := TargetAddress;

CASE TargetAddress OF
    E_RobotAddress.Address01..E_RobotAddress.Address06:
        _Address.nInt := TargetAddress;
ELSE
    Error  := TRUE;
    ErrMsg := 'ClampA target address out of range';
	RETURN;
END_CASE

// Check ClampA Action is correct
CASE ClampAction OF
	E_ClampAction.PickUp:
		_DO3.bGet := TRUE;
	E_ClampAction.Place:
		_DO3.bGet := FALSE;
ELSE
	Error := TRUE;
	ErrMsg := 'ClampA Action is wrong command';
	RETURN;
END_CASE

// Send robot target area data
_DO3.nArea1 := _Area.BitList.Bit0;
_DO3.nArea2 := _Area.BitList.Bit1;
_DO3.nArea3 := _Area.BitList.Bit2;
_DO3.nArea4 := _Area.BitList.Bit3;

// Send robot target address data
_DO3.nAddress1 := _Address.BitList.Bit0;
_DO3.nAddress2 := _Address.BitList.Bit1;
_DO3.nAddress3 := _Address.BitList.Bit2;
_DO3.nAddress4 := _Address.BitList.Bit3;
_DO3.nAddress5 := _Address.BitList.Bit4;
_DO3.nAddress6 := _Address.BitList.Bit5;
_DO3.nAddress7 := _Address.BitList.Bit6;


_DO3.bExecute := NOT Error;

_DO3.bContinue := BoxReady;

M_StartAbsMoveAction_ClampA := NOT Error; // Method end
END_METHOD

(* This Method is used to send command data to Fanuc Robot, only clampB is work 
*)
METHOD M_StartAbsMoveAction_ClampB : BOOL
VAR_INPUT
    TargetArea    : E_RobotArea;    // Select the zone where robot will going.
    TargetAddress : E_RobotAddress; // Because the address num in different zone, the number define is different. But also need >= 1, 0 = undefined
    ClampAction   : E_ClampAction;  // need to define the command
    BoxReady      : BOOL;           // Fanuc robot prog will stop at a safe position just before reaching the target location, until `AllowContinue` is set to true.
END_VAR

VAR_OUTPUT
    Error  : BOOL;
    ErrMsg : T_MaxString;
END_VAR

VAR_INST
    _Area    : ST_IntToBool;
    _Address : ST_IntToBool;
END_VAR
// Set target area
_Area.nInt := TargetArea;

// Check ClampB target area is correct
CASE TargetArea OF
    E_RobotArea.RoundBelt..E_RobotArea.PullOutConveyor:
        _Area.nInt := TargetArea;
ELSE
    Error  := TRUE;
    ErrMsg := 'ClampB target area out of range';
	RETURN;
END_CASE

// Check ClampB target address is correct
CASE TargetAddress OF
	E_RobotAddress.Address01..E_RobotAddress.Address06:
		_Address.nInt := TargetAddress;
ELSE
	Error := TRUE;
	ErrMsg := 'ClampB target address is out of range';
	RETURN;
END_CASE

// Check ClampB Action is correct
CASE ClampAction OF
	E_ClampAction.PickUp:
		_DO4.bGet := TRUE;
	E_ClampAction.Place:
		_DO4.bGet := FALSE;
ELSE
	Error := TRUE;
	ErrMsg := 'ClampB Action is wrong command';
	RETURN;
END_CASE

// Send robot target area data
_DO4.nArea1 := _Area.BitList.Bit0;
_DO4.nArea2 := _Area.BitList.Bit1;
_DO4.nArea3 := _Area.BitList.Bit2;
_DO4.nArea4 := _Area.BitList.Bit3;

// Send robot target address data
_DO4.nAddress1 := _Address.BitList.Bit0;
_DO4.nAddress2 := _Address.BitList.Bit1;
_DO4.nAddress3 := _Address.BitList.Bit2;
_DO4.nAddress4 := _Address.BitList.Bit3;
_DO4.nAddress5 := _Address.BitList.Bit4;
_DO4.nAddress6 := _Address.BitList.Bit5;
_DO4.nAddress7 := _Address.BitList.Bit6;

_DO4.bExecute := NOT Error;

_DO4.bContinue := BoxReady;

M_StartAbsMoveAction_ClampB := NOT Error; // Method end
END_METHOD

METHOD M_StartAbsMoveAction_ClampBoth : BOOL
VAR_INPUT
    ClampA_TargetArea    : E_RobotArea;
    ClampA_TargetAddress : E_RobotAddress;
    ClampA_Action        : E_ClampAction;
    ClampB_TargetArea    : E_RobotArea;
    ClampB_TargetAddress : E_RobotAddress;
    ClampB_Action        : E_ClampAction;
    BoxReady_1st         : BOOL;
    BoxReady_2nd         : BOOL;
END_VAR

VAR_OUTPUT
    Error  : BOOL;
    ErrMsg : T_MaxString;
END_VAR

VAR_INST
    _ClampA_Area    : ST_IntToBool;
    _ClampB_Area    : ST_IntToBool;
    _ClampA_Address : ST_IntToBool;
    _ClampB_Address : ST_IntToBool;
END_VAR
// Set Target Area
_ClampA_Area.nInt := ClampA_TargetArea;
_ClampB_Area.nInt := ClampB_TargetArea;
// Check ClampA target area is correct
CASE ClampA_TargetArea OF
    E_RobotArea.RoundBelt..E_RobotArea.PullOutConveyor:
        _ClampA_Area.nInt := ClampA_TargetArea;
ELSE
    Error  := TRUE;
    ErrMsg := 'ClampA target area out of range';
	RETURN;
END_CASE
// Check ClampA target address is correct
CASE ClampA_TargetAddress OF
    E_RobotAddress.Address01..E_RobotAddress.Address06:
        _ClampA_Address.nInt := ClampA_TargetAddress;
ELSE
    Error  := TRUE;
    ErrMsg := 'ClampA target address out of range';
	RETURN;
END_CASE

// Check ClampA Action is correct
CASE ClampA_Action OF
	E_ClampAction.PickUp:
		_DO3.bGet := TRUE;
	E_ClampAction.Place:
		_DO3.bGet := FALSE;
ELSE
	Error := TRUE;
	ErrMsg := 'ClampA Action is wrong command';
	RETURN;
END_CASE
// Check ClampB target area is correct
CASE ClampB_TargetArea OF
    E_RobotArea.RoundBelt..E_RobotArea.PullOutConveyor:
        _ClampB_Area.nInt := ClampB_TargetArea;
ELSE
	Error := TRUE;
	ErrMsg := 'ClampB target area out of range';
	RETURN;
END_CASE

// Check ClampB target address is correct
CASE ClampB_TargetAddress OF
	E_RobotAddress.Address01..E_RobotAddress.Address06:
		_ClampB_Address.nInt := ClampB_TargetAddress;
ELSE
	Error := TRUE;
	ErrMsg := 'ClampB target address is out of range';
	RETURN;
END_CASE
// Check ClampB Action is correct
CASE ClampB_Action OF
	E_ClampAction.PickUp:
		_DO4.bGet := TRUE;
	E_ClampAction.Place:
		_DO4.bGet := FALSE;
ELSE
	Error := TRUE;
	ErrMsg := 'ClampB Action is wrong command';
	RETURN;
END_CASE

// Send robot target area data
_DO3.nArea1 := _ClampA_Area.BitList.Bit0;
_DO3.nArea2 := _ClampA_Area.BitList.Bit1;
_DO3.nArea3 := _ClampA_Area.BitList.Bit2;
_DO3.nArea4 := _ClampA_Area.BitList.Bit3;

_DO4.nArea1 := _ClampB_Area.BitList.Bit0;
_DO4.nArea2 := _ClampB_Area.BitList.Bit1;
_DO4.nArea3 := _ClampB_Area.BitList.Bit2;
_DO4.nArea4 := _ClampB_Area.BitList.Bit3;

// Send robot target address data
_DO3.nAddress1 := _ClampA_Address.BitList.Bit0;
_DO3.nAddress2 := _ClampA_Address.BitList.Bit1;
_DO3.nAddress3 := _ClampA_Address.BitList.Bit2;
_DO3.nAddress4 := _ClampA_Address.BitList.Bit3;
_DO3.nAddress5 := _ClampA_Address.BitList.Bit4;
_DO3.nAddress6 := _ClampA_Address.BitList.Bit5;
_DO3.nAddress7 := _ClampA_Address.BitList.Bit6;

_DO4.nAddress1 := _ClampB_Address.BitList.Bit0;
_DO4.nAddress2 := _ClampB_Address.BitList.Bit1;
_DO4.nAddress3 := _ClampB_Address.BitList.Bit2;
_DO4.nAddress4 := _ClampB_Address.BitList.Bit3;
_DO4.nAddress5 := _ClampB_Address.BitList.Bit4;
_DO4.nAddress6 := _ClampB_Address.BitList.Bit5;
_DO4.nAddress7 := _ClampB_Address.BitList.Bit6;

_DO3.bExecute := NOT Error;
_DO4.bExecute := NOT Error;

_DO3.bContinue := BoxReady_1st;
_DO4.bContinue := BoxReady_2nd;

M_StartAbsMoveAction_ClampBoth := NOT Error; // Method end
END_METHOD

METHOD M_StartMoveBoxToFeedInConveyor_ClampA : BOOL
VAR_INPUT
    ConveyorSlideSelect : E_FeedInEmptyBox_PlaceArea;
    DiffSizeSlideClear  : BOOL;
    SameSizeSlideClear  : BOOL;
END_VAR
VAR_INST
    _Area    : ST_IntToBool;
    _Address : ST_IntToBool;
END_VAR
// Set target area is round belt
_Area.nInt := E_RobotArea.TransmitCV;
IF ConveyorSlideSelect = E_FeedInEmptyBox_PlaceArea.DiffSizeConveyor THEN
	_Address.nInt := 1;
ELSIF ConveyorSlideSelect = E_FeedInEmptyBox_PlaceArea.SameSizeConveyor THEN
	_Address.nInt := 2;
ELSE
	// Wrong command, return
	RETURN ;
END_IF
// Send robot target area data
_DO3.nArea1 := _Area.BitList.Bit0;
_DO3.nArea2 := _Area.BitList.Bit1;
_DO3.nArea3 := _Area.BitList.Bit2;
_DO3.nArea4 := _Area.BitList.Bit3;

// Send robot target address data
_DO3.nAddress1 := _Address.BitList.Bit0;
_DO3.nAddress2 := _Address.BitList.Bit1;
_DO3.nAddress3 := _Address.BitList.Bit2;
_DO3.nAddress4 := _Address.BitList.Bit3;
_DO3.nAddress5 := _Address.BitList.Bit4;
_DO3.nAddress6 := _Address.BitList.Bit5;
_DO3.nAddress7 := _Address.BitList.Bit6;

_DO3.bGet := FALSE; // Place action

_DO3.bExecute := TRUE;
IF ConveyorSlideSelect = E_FeedInEmptyBox_PlaceArea.DiffSizeConveyor THEN
	_DO3.bContinue := DiffSizeSlideClear;
ELSIF ConveyorSlideSelect = E_FeedInEmptyBox_PlaceArea.SameSizeConveyor THEN
	_DO3.bContinue := SameSizeSlideClear;
END_IF
M_StartMoveBoxToFeedInConveyor_ClampA := TRUE ; // Method end
END_METHOD

METHOD M_StartMoveBoxToFeedInConveyor_ClampB : BOOL
VAR_INPUT
	ConveyorSlideSelect : E_FeedInEmptyBox_PlaceArea;
    DiffSizeSlideClear  : BOOL;
    SameSizeSlideClear  : BOOL;
END_VAR
VAR_INST
	_Area : ST_IntToBool;
	_Address_ClampB :ST_IntToBool;
END_VAR
// Set target area is round belt
_Area.nInt := E_RobotArea.TransmitCV;
IF ConveyorSlideSelect = E_FeedInEmptyBox_PlaceArea.DiffSizeConveyor THEN
	_Address_ClampB.nInt := 1;
ELSIF ConveyorSlideSelect = E_FeedInEmptyBox_PlaceArea.SameSizeConveyor THEN
	_Address_ClampB.nInt := 2;
ELSE
	// Wrong command, return
	RETURN ;
END_IF
// Send robot target area data
_DO4.nArea1 := _Area.BitList.Bit0;
_DO4.nArea2 := _Area.BitList.Bit1;
_DO4.nArea3 := _Area.BitList.Bit2;
_DO4.nArea4 := _Area.BitList.Bit3;

// Send robot target address data
_DO4.nAddress1 := _Address_ClampB.BitList.Bit0;
_DO4.nAddress2 := _Address_ClampB.BitList.Bit1;
_DO4.nAddress3 := _Address_ClampB.BitList.Bit2;
_DO4.nAddress4 := _Address_ClampB.BitList.Bit3;
_DO4.nAddress5 := _Address_ClampB.BitList.Bit4;
_DO4.nAddress6 := _Address_ClampB.BitList.Bit5;
_DO4.nAddress7 := _Address_ClampB.BitList.Bit6;

_DO4.bGet := FALSE; // Place action

_DO4.bExecute := TRUE;
IF ConveyorSlideSelect = E_FeedInEmptyBox_PlaceArea.DiffSizeConveyor THEN
	_DO4.bContinue := DiffSizeSlideClear;
ELSIF ConveyorSlideSelect = E_FeedInEmptyBox_PlaceArea.SameSizeConveyor THEN
	_DO4.bContinue := SameSizeSlideClear;
END_IF
M_StartMoveBoxToFeedInConveyor_ClampB := TRUE; // Method end
END_METHOD

METHOD M_StartMoveBoxToFeedInConveyor_ClampBoth : BOOL
VAR_INPUT
//    ConveyorSlideSelect : E_FeedInEmptyBox_PlaceArea;
    ClampA_Address      : E_FeedInEmptyBox_PlaceArea;
    ClampB_Address      : E_FeedInEmptyBox_PlaceArea;
	SlideClear_1st : BOOL;
	SlideClear_2nd : BOOL;
END_VAR
VAR_INST
    _Area           : ST_IntToBool;
    _Address_ClampA : ST_IntToBool;
    _Address_ClampB : ST_IntToBool;
END_VAR
// Set target area is round belt
_Area.nInt := E_RobotArea.TransmitCV;
// Select ClampA target address
IF ClampA_Address = E_FeedInEmptyBox_PlaceArea.DiffSizeConveyor THEN
	_Address_ClampA.nInt := 1;
ELSIF ClampA_Address = E_FeedInEmptyBox_PlaceArea.SameSizeConveyor THEN
	_Address_ClampA.nInt := 2;
ELSE
	// Wrong command, return
	RETURN ;
END_IF

// Select ClampB target address
IF ClampB_Address = E_FeedInEmptyBox_PlaceArea.DiffSizeConveyor THEN
	_Address_ClampB.nInt := 1;
ELSIF ClampB_Address = E_FeedInEmptyBox_PlaceArea.SameSizeConveyor THEN
	_Address_ClampB.nInt := 2;
ELSE
	// Wrong command, return
	RETURN;
END_IF

// Send robot target area data
_DO3.nArea1 := _Area.BitList.Bit0;
_DO3.nArea2 := _Area.BitList.Bit1;
_DO3.nArea3 := _Area.BitList.Bit2;
_DO3.nArea4 := _Area.BitList.Bit3;

_DO4.nArea1 := _Area.BitList.Bit0;
_DO4.nArea2 := _Area.BitList.Bit1;
_DO4.nArea3 := _Area.BitList.Bit2;
_DO4.nArea4 := _Area.BitList.Bit3;

// Send robot clampA target address data
_DO3.nAddress1 := _Address_ClampA.BitList.Bit0;
_DO3.nAddress2 := _Address_ClampA.BitList.Bit1;
_DO3.nAddress3 := _Address_ClampA.BitList.Bit2;
_DO3.nAddress4 := _Address_ClampA.BitList.Bit3;
_DO3.nAddress5 := _Address_ClampA.BitList.Bit4;
_DO3.nAddress6 := _Address_ClampA.BitList.Bit5;
_DO3.nAddress7 := _Address_ClampA.BitList.Bit6;

_do4.nAddress1 := _Address_ClampB.BitList.Bit0;
_do4.nAddress2 := _Address_ClampB.BitList.Bit1;
_do4.nAddress3 := _Address_ClampB.BitList.Bit2;
_do4.nAddress4 := _Address_ClampB.BitList.Bit3;
_do4.nAddress5 := _Address_ClampB.BitList.Bit4;
_do4.nAddress6 := _Address_ClampB.BitList.Bit5;
_do4.nAddress7 := _Address_ClampB.BitList.Bit6;


_DO3.bGet := FALSE;
_DO4.bGet := FALSE;

_DO3.bExecute := TRUE;
_DO4.bExecute := TRUE;

_DO3.bContinue := SlideClear_1st;
_DO4.bContinue := SlideClear_2nd;

M_StartMoveBoxToFeedInConveyor_ClampBoth := TRUE; // Method end
END_METHOD

METHOD M_StartMoveBoxToRoundBelt_Both : BOOL
VAR_INPUT
	CarrierSelect_ClampA : E_ReloadRoundBelt_PlaceAddress;
	CarrierSelect_ClampB : E_ReloadRoundBelt_PlaceAddress;
	A2_Sensor : BOOL;
	A3_Sensor : BOOL;
	RoundBeltSafe_1st : BOOL;
	RoundBeltSafe_2nd : BOOL;
END_VAR
VAR_INST
	_Area1 : ST_IntToBool;
	_Address1 : ST_IntToBool;
	CarrierAddress1 :E_ReloadRoundBelt_PlaceAddress;
	_Area2: ST_IntToBool;
	_Address2 : ST_IntToBool;
	CarrierAddress2 :E_ReloadRoundBelt_PlaceAddress;
END_VAR
// Set target area is round belt
_Area1.nInt := E_RobotArea.RoundBelt;
_Area2.nInt := E_RobotArea.RoundBelt;

IF CarrierSelect_ClampA = E_ReloadRoundBelt_PlaceAddress.A2 THEN
	_Address1.nInt := 1;
ELSIF CarrierSelect_ClampA = E_ReloadRoundBelt_PlaceAddress.A3 THEN
	_Address1.nInt := 2;
ELSE
	// Wrong command, return
	RETURN;
END_IF

IF CarrierSelect_ClampB = E_ReloadRoundBelt_PlaceAddress.A2 THEN
	_Address2.nInt := 1;
ELSIF CarrierSelect_ClampB = E_ReloadRoundBelt_PlaceAddress.A3 THEN
	_Address2.nInt := 2;
ELSE
	// Wrong command return
	RETURN;
END_IF
// Send robot target area data
_DO3.nArea1 := _Area1.BitList.Bit0;
_DO3.nArea2 := _Area1.BitList.Bit1;
_DO3.nArea3 := _Area1.BitList.Bit2;
_DO3.nArea4 := _Area1.BitList.Bit3;

_DO4.nArea1 := _Area2.BitList.Bit0;
_DO4.nArea2 := _Area2.BitList.Bit1;
_DO4.nArea3 := _Area2.BitList.Bit2;
_DO4.nArea4 := _Area2.BitList.Bit3;

// Send robot target address data
_DO3.nAddress1 := _Address1.BitList.Bit0;
_DO3.nAddress2 := _Address1.BitList.Bit1;
_DO3.nAddress3 := _Address1.BitList.Bit2;
_DO3.nAddress4 := _Address1.BitList.Bit3;
_DO3.nAddress5 := _Address1.BitList.Bit4;
_DO3.nAddress6 := _Address1.BitList.Bit5;
_DO3.nAddress7 := _Address1.BitList.Bit6;

_DO4.nAddress1 := _Address2.BitList.Bit0;
_DO4.nAddress2 := _Address2.BitList.Bit1;
_DO4.nAddress3 := _Address2.BitList.Bit2;
_DO4.nAddress4 := _Address2.BitList.Bit3;
_DO4.nAddress5 := _Address2.BitList.Bit4;
_DO4.nAddress6 := _Address2.BitList.Bit5;
_DO4.nAddress7 := _Address2.BitList.Bit6;

_DO3.bGet := FALSE; // ClampA Place action
_DO4.bGet := FALSE; // ClampB Place action

IF CarrierSelect_ClampA = E_ReloadRoundBelt_PlaceAddress.A2 THEN
	_DO3.bContinue := NOT A2_Sensor AND RoundBeltSafe_1st;
ELSIF 	CarrierSelect_ClampA = E_ReloadRoundBelt_PlaceAddress.A3 THEN
	_DO3.bContinue := NOT A3_Sensor AND RoundBeltSafe_1st;
END_IF

IF CarrierSelect_ClampB = E_ReloadRoundBelt_PlaceAddress.A2 THEN
	_DO4.bContinue := NOT A2_Sensor AND RoundBeltSafe_2nd;
ELSIF CarrierSelect_ClampB = E_ReloadRoundBelt_PlaceAddress.A3 THEN
	_DO4.bContinue := NOT A3_Sensor AND RoundBeltSafe_2nd;
END_IF

_DO3.bExecute := TRUE; // ClampA Place action
_DO4.bExecute := TRUE; // ClampB Place action


M_StartMoveBoxToRoundBelt_Both := TRUE; // Method end
END_METHOD

METHOD M_StartMoveBoxToRoundBelt_ClampA : BOOL
VAR_INPUT
    CarrierSelect : E_ReloadRoundBelt_PlaceAddress;
    A2_Sensor     : BOOL;
    A3_Sensor     : BOOL;
	RoundBeltSafe : BOOL;
END_VAR
VAR_INST
    _Area          : ST_IntToBool;
    _Address       : ST_IntToBool;
    CarrierAddress : E_ReloadRoundBelt_PlaceAddress;
END_VAR
// Set target area is round belt
_Area.nInt := E_RobotArea.RoundBelt;

IF CarrierSelect = E_ReloadRoundBelt_PlaceAddress.A2 THEN
    _Address.nInt := 1;
ELSIF CarrierSelect = E_ReloadRoundBelt_PlaceAddress.A3 THEN
    _Address.nInt := 2;
ELSE
    // Wrong command, return
    RETURN;
END_IF

// Send robot target area data
_DO3.nArea1 := _Area.BitList.Bit0;
_DO3.nArea2 := _Area.BitList.Bit1;
_DO3.nArea3 := _Area.BitList.Bit2;
_DO3.nArea4 := _Area.BitList.Bit3;

// Send robot target address data
_DO3.nAddress1 := _Address.BitList.Bit0;
_DO3.nAddress2 := _Address.BitList.Bit1;
_DO3.nAddress3 := _Address.BitList.Bit2;
_DO3.nAddress4 := _Address.BitList.Bit3;
_DO3.nAddress5 := _Address.BitList.Bit4;
_DO3.nAddress6 := _Address.BitList.Bit5;
_DO3.nAddress7 := _Address.BitList.Bit6;

_DO3.bGet := FALSE; // Place action

_DO3.bExecute := TRUE;

IF CarrierSelect = E_ReloadRoundBelt_PlaceAddress.A2 THEN
    _DO3.bContinue := NOT A2_Sensor AND RoundBeltSafe ; // Carrier A2 did not has box
ELSIF CarrierSelect = E_ReloadRoundBelt_PlaceAddress.A3 THEN
    _DO3.bContinue := NOT A3_Sensor AND RoundBeltSafe; // Carrier A3 did not has box
END_IF

M_StartMoveBoxToRoundBelt_ClampA := true; // Method end
END_METHOD

METHOD M_StartMoveBoxToRoundBelt_ClampB : BOOL
VAR_INPUT
    CarrierSelect : E_ReloadRoundBelt_PlaceAddress;
    A2_Sensor     : BOOL;
    A3_Sensor     : BOOL;
	RoundBeltSafe : BOOL;
END_VAR
VAR_INST
    _Area          : ST_IntToBool;
    _Address       : ST_IntToBool;
    CarrierAddress : E_ReloadRoundBelt_PlaceAddress;
END_VAR
// Set target area is round belt
_Area.nInt := E_RobotArea.RoundBelt;
IF CarrierSelect = E_ReloadRoundBelt_PlaceAddress.A2 THEN
	_Address.nInt := 1;
ELSIF  CarrierSelect = E_ReloadRoundBelt_PlaceAddress.A3 THEN
	_Address.nInt := 2;
ELSE
	// Wrong command, return
	RETURN ;
END_IF

// Send robot target area data
_DO4.nArea1 := _Area.BitList.Bit0;
_DO4.nArea2 := _Area.BitList.Bit1;
_DO4.nArea3 := _Area.BitList.Bit2;
_DO4.nArea4 := _Area.BitList.Bit3;

// Send robot target address data
_DO4.nAddress1 := _Address.BitList.Bit0;
_DO4.nAddress2 := _Address.BitList.Bit1;
_DO4.nAddress3 := _Address.BitList.Bit2;
_DO4.nAddress4 := _Address.BitList.Bit3;
_DO4.nAddress5 := _Address.BitList.Bit4;
_DO4.nAddress6 := _Address.BitList.Bit5;
_DO4.nAddress7 := _Address.BitList.Bit6;

_DO4.bGet := FALSE; // Place action

_DO4.bExecute := TRUE;

IF CarrierSelect = E_ReloadRoundBelt_PlaceAddress.A2 THEN
	_DO4.bContinue := NOT A2_Sensor AND RoundBeltSafe; // Carrier A2 did not has box
ELSIF CarrierSelect = E_ReloadRoundBelt_PlaceAddress.A3 THEN
	_DO4.bContinue := NOT A3_Sensor AND RoundBeltSafe; // Carrier A3 did not has box
END_IF

M_StartMoveBoxToRoundBelt_ClampB := TRUE; // Method end
END_METHOD

(* This method is used to setting the Fanuc Robot Action " Pickup box from PulloutConveyor , only clampA"
*)
METHOD M_StartPullOutConveyorPickUpBox_ClampA : BOOL
VAR_INPUT
	ClampA_Address : E_PullOutConveyorPosition;
	BoxReady : BOOL; // True : Pullout conveyor box is ready. accroding ClampA target slide is ready or not.
END_VAR
VAR_INST
	_Area : ST_IntToBool;
    _Address_ClampA : ST_IntToBool;
END_VAR
// Set target area is round belt
_Area.nInt := E_RobotArea.PullOutConveyor;
// Select pullout conveyor slide
IF ClampA_Address = E_PullOutConveyorPosition.I3_Slide THEN
	_Address_ClampA.nInt := 1;
ELSIF ClampA_Address = E_PullOutConveyorPosition.I4_Slide THEN
	_Address_ClampA.nInt := 2;
ELSE
	// Wrong command, return
	RETURN ;
END_IF
// Send robot target area data
_DO3.nArea1 := _Area.BitList.Bit0;
_DO3.nArea2 := _Area.BitList.Bit1;
_DO3.nArea3 := _Area.BitList.Bit2;
_DO3.nArea4 := _Area.BitList.Bit3;

// Send robot target address data
_DO3.nAddress1 := _Address_ClampA.BitList.Bit0;
_DO3.nAddress2 := _Address_ClampA.BitList.Bit1;
_DO3.nAddress3 := _Address_ClampA.BitList.Bit2;
_DO3.nAddress4 := _Address_ClampA.BitList.Bit3;
_DO3.nAddress5 := _Address_ClampA.BitList.Bit4;
_DO3.nAddress6 := _Address_ClampA.BitList.Bit5;
_DO3.nAddress7 := _Address_ClampA.BitList.Bit6;

_DO3.bGet := TRUE; // Pickup action
_DO3.bExecute := TRUE;

_DO3.bContinue := BoxReady;

M_StartPullOutConveyorPickUpBox_ClampA := true; // Method end
END_METHOD

(* This method is used to setting the Fanuc Robot Action " Pickup box from PulloutConveyor , only clampB"
*)
METHOD M_StartPullOutConveyorPickUpBox_ClampB : BOOL
VAR_INPUT
	ClampB_Address :E_PullOutConveyorPosition;
	BoxReady : BOOL; // True : Pullout conveyor box is ready. accroding ClampA target slide is ready or not.
END_VAR
VAR_INST
	_Area : ST_IntToBool;
    _Address_ClampB : ST_IntToBool;
END_VAR
// Set target area is round belt
_Area.nInt := E_RobotArea.PullOutConveyor;
// Select pullout conveyor slide
IF ClampB_Address = E_PullOutConveyorPosition.I3_Slide THEN
	_Address_ClampB.nInt := 1;
ELSIF ClampB_Address = E_PullOutConveyorPosition.I4_Slide THEN
	_Address_ClampB.nInt := 2;
ELSE
	// Wrong command, return
	RETURN ;
END_IF

// Send robot target area data
_DO4.nArea1 := _Area.BitList.Bit0;
_DO4.nArea2 := _Area.BitList.Bit1;
_DO4.nArea3 := _Area.BitList.Bit2;
_DO4.nArea4 := _Area.BitList.Bit3;

// Send robot target address data
_DO4.nAddress1 := _Address_ClampB.BitList.Bit0;
_DO4.nAddress2 := _Address_ClampB.BitList.Bit1;
_DO4.nAddress3 := _Address_ClampB.BitList.Bit2;
_DO4.nAddress4 := _Address_ClampB.BitList.Bit3;
_DO4.nAddress5 := _Address_ClampB.BitList.Bit4;
_DO4.nAddress6 := _Address_ClampB.BitList.Bit5;
_DO4.nAddress7 := _Address_ClampB.BitList.Bit6;

_DO4.bGet := TRUE; // Pickup action
_DO4.bExecute := TRUE;

_DO4.bContinue := BoxReady;

M_StartPullOutConveyorPickUpBox_ClampB := true; // Method end
END_METHOD

(* This method is used to setting the Fanuc Robot Action " Pickup box from PulloutConveyor, both clamp"
*)
METHOD M_StartPullOutConveyorPickUpBox_ClampBoth : BOOL
VAR_INPUT
	ClampA_Address : E_PullOutConveyorPosition;
	ClampB_Address : E_PullOutConveyorPosition;
	BoxReady_1 : BOOL; // TRUE : 1st target slide box is ready
	BoxReady_2 : BOOL; // True : 2nd target slide box is ready
END_VAR
VAR_INST
	_Area : ST_IntToBool;
    _Address_ClampA : ST_IntToBool;
    _Address_ClampB : ST_IntToBool;
END_VAR
// Set target area is round belt
_Area.nInt := E_RobotArea.PullOutConveyor;

// Select ClampA target address
IF ClampA_Address = E_PullOutConveyorPosition.I3_Slide THEN
    _Address_ClampA.nInt := 1;
ELSIF ClampA_Address = E_PullOutConveyorPosition.I4_Slide THEN
    _Address_ClampA.nInt := 2;
ELSE
    // Wrong command, return
    RETURN;
END_IF

// Select ClampB target address
IF ClampB_Address = E_PullOutConveyorPosition.I3_Slide THEN
    _Address_ClampB.nInt := 1;
ELSIF ClampB_Address = E_PullOutConveyorPosition.I4_Slide THEN
    _Address_ClampB.nInt := 2;
ELSE
    // Wrong command, return
    RETURN;
END_IF

// Send robot target area data
_DO3.nArea1 := _Area.BitList.Bit0;
_DO3.nArea2 := _Area.BitList.Bit1;
_DO3.nArea3 := _Area.BitList.Bit2;
_DO3.nArea4 := _Area.BitList.Bit3;

_DO4.nArea1 := _Area.BitList.Bit0;
_DO4.nArea2 := _Area.BitList.Bit1;
_DO4.nArea3 := _Area.BitList.Bit2;
_DO4.nArea4 := _Area.BitList.Bit3;

// Send robot target address data
_DO3.nAddress1 := _Address_ClampA.BitList.Bit0;
_DO3.nAddress2 := _Address_ClampA.BitList.Bit1;
_DO3.nAddress3 := _Address_ClampA.BitList.Bit2;
_DO3.nAddress4 := _Address_ClampA.BitList.Bit3;
_DO3.nAddress5 := _Address_ClampA.BitList.Bit4;
_DO3.nAddress6 := _Address_ClampA.BitList.Bit5;
_DO3.nAddress7 := _Address_ClampA.BitList.Bit6;

_DO4.nAddress1 := _Address_ClampB.BitList.Bit0;
_DO4.nAddress2 := _Address_ClampB.BitList.Bit1;
_DO4.nAddress3 := _Address_ClampB.BitList.Bit2;
_DO4.nAddress4 := _Address_ClampB.BitList.Bit3;
_DO4.nAddress5 := _Address_ClampB.BitList.Bit4;
_DO4.nAddress6 := _Address_ClampB.BitList.Bit5;
_DO4.nAddress7 := _Address_ClampB.BitList.Bit6;

_DO3.bGet := TRUE;
_DO4.bGet := TRUE;

_DO3.bExecute := TRUE;
_DO4.bExecute := TRUE;

_DO3.bContinue := BoxReady_1;
_DO4.bContinue := BoxReady_2;

M_StartPullOutConveyorPickUpBox_ClampBoth := true; // Method end
END_METHOD

METHOD PUBLIC M_StartRobotAbsMove : BOOL
VAR_INPUT
	GetBox		: BOOL;
	UseClampA	: BOOL;
	UseClampB   : BOOL;
	Area : E_RobotArea;
	
	
	ClampA_Address	: INT;
	ClampB_Address	: INT;

	BoxReady_1 : BOOL;
	BoxReady_2 : BOOL;
	
END_VAR

VAR_INST
	_Area	: ST_IntToBool;
	_Address_ClampA : ST_IntToBool;
    _Address_ClampB : ST_IntToBool;
END_VAR
//Set target area
_Area.nInt :=Area;

IF UseClampA THEN
	_Address_ClampA.nInt:=ClampA_Address;
	_DO3.nArea1 := _Area.BitList.Bit0;
	_DO3.nArea2 := _Area.BitList.Bit1;
	_DO3.nArea3 := _Area.BitList.Bit2;
	_DO3.nArea4 := _Area.BitList.Bit3;

	_DO3.nAddress1 := _Address_ClampA.BitList.Bit0;
	_DO3.nAddress2 := _Address_ClampA.BitList.Bit1;
	_DO3.nAddress3 := _Address_ClampA.BitList.Bit2;
	_DO3.nAddress4 := _Address_ClampA.BitList.Bit3;
	_DO3.nAddress5 := _Address_ClampA.BitList.Bit4;
	_DO3.nAddress6 := _Address_ClampA.BitList.Bit5;
	_DO3.nAddress7 := _Address_ClampA.BitList.Bit6;
	_DO3.bGet := GetBox;
	_DO3.bExecute := TRUE;
	_DO3.bContinue := BoxReady_1;	
END_IF

IF UseClampB THEN
	_Address_ClampB.nInt:=ClampB_Address;
	_DO4.nArea1 := _Area.BitList.Bit0;
	_DO4.nArea2 := _Area.BitList.Bit1;
	_DO4.nArea3 := _Area.BitList.Bit2;
	_DO4.nArea4 := _Area.BitList.Bit3;
	
	_DO4.nAddress1 := _Address_ClampB.BitList.Bit0;
	_DO4.nAddress2 := _Address_ClampB.BitList.Bit1;
	_DO4.nAddress3 := _Address_ClampB.BitList.Bit2;
	_DO4.nAddress4 := _Address_ClampB.BitList.Bit3;
	_DO4.nAddress5 := _Address_ClampB.BitList.Bit4;
	_DO4.nAddress6 := _Address_ClampB.BitList.Bit5;
	_DO4.nAddress7 := _Address_ClampB.BitList.Bit6;
	_DO4.bGet := GetBox;
	_DO4.bExecute := TRUE;
	_DO4.bContinue := BoxReady_2;	
END_IF

M_StartRobotAbsMove :=TRUE;




















M_StartRobotAbsMove:=TRUE;
END_METHOD

METHOD M_StartWarehouseMoveAction_ClampA : BOOL
VAR_INPUT
	WareHouseSelect : E_WareHouse;
	Info : ST_WareHouseCoordinates; // Input Warehouse with robot move parameter for pickup box;
	ClampAction :E_ClampAction;
	BoxReady : BOOL;
END_VAR
VAR_OUTPUT
	Error : BOOL;
	ErrMsg :T_MaxString;
END_VAR
VAR_INST
	_Layer : ST_IntToBool;
	_Slide : ST_IntToBool;
END_VAR
// Set target warehouse
CASE WareHouseSelect OF
    E_WareHouse.WareHouseA:
        _DO1.bTargetWareHouseA := TRUE;
        _DO1.bTargetWareHouseB := FALSE;
    E_WareHouse.WareHouseB:
        _DO1.bTargetWareHouseA := FALSE;
        _DO1.bTargetWareHouseB := TRUE;
ELSE
    _DO1.bTargetWareHouseA := FALSE;
    _DO1.bTargetWareHouseB := FALSE;
    Error                  := TRUE;
    ErrMsg                 := 'ClampA target warehouse out of range';
	RETURN;
END_CASE

// Set Warehouse coordinates
_Layer.nInt := info.Layer;
_Slide.nInt := info.Slide;

// Send Layer data to robot
_DO1.nLayer1 := _Layer.BitList.Bit0;
_DO1.nLayer2 := _Layer.BitList.Bit1;
_DO1.nLayer3 := _Layer.BitList.Bit2;
_DO1.nLayer4 := _Layer.BitList.Bit3;

// Send Slide data to Robot
_DO1.nSlide1 := _Slide.BitList.Bit0;
_DO1.nSlide2 := _Slide.BitList.Bit1;
_DO1.nSlide3 := _Slide.BitList.Bit2;
_DO1.nSlide4 := _Slide.BitList.Bit3;
_DO1.nSlide5 := _Slide.BitList.Bit4;

// Send clamp action to robot
CASE ClampAction OF
	E_ClampAction.PickUp:
		_DO1.bGet := TRUE;
	E_ClampAction.Place:
		_DO1.bGet := FALSE;
ELSE
	Error := TRUE;
	ErrMsg := 'Clamp action not defined';
	RETURN;
END_CASE

// Send action data to robot
_DO1.bExecute := NOT Error;
_DO1.bContinue := BoxReady;
M_StartWarehouseMoveAction_ClampA := NOT Error; // Method end
END_METHOD

METHOD M_StartWarehouseMoveAction_ClampB : BOOL
VAR_INPUT
	WareHouseSelect : E_WareHouse;
	Info : ST_WareHouseCoordinates; // Input Warehouse with robot move parameter for pickup box;
	ClampAction :E_ClampAction;
	BoxReady : BOOL;
END_VAR
VAR_OUTPUT
	Error : BOOL;
	ErrMsg :T_MaxString;
END_VAR
VAR_INST
	_Layer : ST_IntToBool;
	_Slide : ST_IntToBool;
END_VAR
// Set target warehouse
CASE WareHouseSelect OF
    E_WareHouse.WareHouseA:
        _DO2.bTargetWareHouseA := TRUE;
        _DO2.bTargetWareHouseB := FALSE;
    E_WareHouse.WareHouseB:
        _DO2.bTargetWareHouseA := FALSE;
        _DO2.bTargetWareHouseB := TRUE;
ELSE
    _DO2.bTargetWareHouseA := FALSE;
    _DO2.bTargetWareHouseB := FALSE;
    Error                  := TRUE;
    ErrMsg                 := 'ClampB target warehouse out of range';
	RETURN;
END_CASE

// Set Warehouse coordinates
_Layer.nInt := info.Layer;
_Slide.nInt := info.Slide;

// Send Layer data to robot
_DO2.nLayer1 := _Layer.BitList.Bit0;
_DO2.nLayer2 := _Layer.BitList.Bit1;
_DO2.nLayer3 := _Layer.BitList.Bit2;
_DO2.nLayer4 := _Layer.BitList.Bit3;

// Send Slide data to Robot
_DO2.nSlide1 := _Slide.BitList.Bit0;
_DO2.nSlide2 := _Slide.BitList.Bit1;
_DO2.nSlide3 := _Slide.BitList.Bit2;
_DO2.nSlide4 := _Slide.BitList.Bit3;
_DO2.nSlide5 := _Slide.BitList.Bit4;

// Send clamp action to robot
CASE ClampAction OF
	E_ClampAction.PickUp:
		_DO2.bGet := TRUE;
	E_ClampAction.Place:
		_DO2.bGet := FALSE;
ELSE
	Error := TRUE;
	ErrMsg := 'Clamp action not defined';
	RETURN;
END_CASE

// Send action data to robot
_DO2.bExecute := NOT Error;
_DO2.bContinue := BoxReady;

M_StartWarehouseMoveAction_ClampB := NOT Error; // Method End
END_METHOD

METHOD M_StartWarehouseMoveAction_ClampBoth : BOOL
VAR_INPUT
	WareHouseSelect : E_WareHouse;
	ClampA_Info : ST_WareHouseCoordinates; // Input Warehouse with robot move parameter for pickup box;
	ClampB_Info : ST_WareHouseCoordinates; // Input Warehouse with robot move parameter for pickup box;
	ClampAction_A : E_ClampAction;
	ClampAction_B : E_ClampAction;
	BoxReady_1st : BOOL; // Box is arrived, ready to pickup
	BoxReady_2nd : BOOL; // Box is arrived, ready to pickup
END_VAR
VAR_OUTPUT
	Error : BOOL;
	ErrMsg :T_MaxString;
END_VAR
VAR_INST
	_LayerClampA :ST_IntToBool;
	_SlideClampA : ST_IntToBool;
	_LayerClampB : ST_IntToBool;
	_SLideClampB : ST_IntToBool;
END_VAR
// Set target warehouse
CASE WareHouseSelect OF
    E_WareHouse.WareHouseA:
        _DO1.bTargetWareHouseA := TRUE;
        _DO1.bTargetWareHouseB := FALSE;
        _DO2.bTargetWareHouseA := TRUE;
        _DO2.bTargetWareHouseB := FALSE;
    E_WareHouse.WareHouseB:
        _DO1.bTargetWareHouseA := FALSE;
        _DO1.bTargetWareHouseB := TRUE;
        _DO2.bTargetWareHouseA := FALSE;
        _DO2.bTargetWareHouseB := TRUE;
ELSE
    _DO1.bTargetWareHouseA := FALSE;
    _DO1.bTargetWareHouseB := FALSE;
    _DO2.bTargetWareHouseA := FALSE;
    _DO2.bTargetWareHouseB := FALSE;
    Error                  := TRUE;
    ErrMsg                 := 'Clamp target warehouse out of range';
    RETURN;
END_CASE

// Assign coordinates 
_LayerClampA.nInt := ClampA_Info.Layer;
_SlideClampA.nInt := ClampA_Info.Slide;
_LayerClampB.nInt := ClampB_Info.Layer;
_SlideClampB.nInt := ClampB_Info.Slide;

// Send Layer data to Robot
_DO1.nLayer1 := _LayerClampA.BitList.Bit0;
_DO1.nLayer2 := _LayerClampA.BitList.Bit1;
_DO1.nLayer3 := _LayerClampA.BitList.Bit2;
_DO1.nLayer4 := _LayerClampA.BitList.Bit3;
_DO2.nLayer1 := _LayerClampB.BitList.Bit0;
_DO2.nLayer2 := _LayerClampB.BitList.Bit1;
_DO2.nLayer3 := _LayerClampB.BitList.Bit2;
_DO2.nLayer4 := _LayerClampB.BitList.Bit3;
// Send Slide data to Robot
_DO1.nSlide1 := _SlideClampA.BitList.Bit0;
_DO1.nSlide2 := _SlideClampA.BitList.Bit1;
_DO1.nSlide3 := _SlideClampA.BitList.Bit2;
_DO1.nSlide4 := _SlideClampA.BitList.Bit3;
_DO1.nSlide5 := _SlideClampA.BitList.Bit4;

_DO2.nSlide1 := _SlideClampB.BitList.Bit0;
_DO2.nSlide2 := _SlideClampB.BitList.Bit1;
_DO2.nSlide3 := _SlideClampB.BitList.Bit2;
_DO2.nSlide4 := _SlideClampB.BitList.Bit3;
_DO2.nSlide5 := _SlideClampB.BitList.Bit4;

// Set clamp action 
CASE ClampAction_A OF
	E_ClampAction.PickUp:
		_DO1.bGet := TRUE;
	E_ClampAction.Place:
		_DO1.bGet := FALSE;
ELSE
	Error := TRUE;
	ErrMsg := 'ClampA action not defined';
	RETURN;
END_CASE

// Set clamp action
CASE ClampAction_B OF
	E_ClampAction.PickUp:
		_DO2.bGet := TRUE;
	E_ClampAction.Place:
		_DO2.bGet := FALSE;
ELSE
	Error := TRUE;
	ErrMsg := 'ClampB action not defined';
	RETURN;	
END_CASE

// set execute
_DO1.bExecute := NOT Error;
_DO2.bExecute := NOT Error;

_DO1.bContinue := BoxReady_1st;
_DO2.bContinue := BoxReady_2nd;

M_StartWarehouseMoveAction_ClampBoth := NOT Error; // Method end
END_METHOD

METHOD M_StartWareHousePickUpBox_ClampA : Bool
VAR_INPUT
	WareHouseSelect : E_WareHouse;
	Info : ST_WareHouseCoordinates; // Input Warehouse with robot move parameter for pickup box;
	BoxReady_1st : BOOL;
END_VAR
VAR_INST
	_Layer : ST_IntToBool;
	_Slide : ST_IntToBool;
END_VAR
// Send target warehouse to robot
IF WareHouseSelect = E_WareHouse.WareHouseA THEN
	_DO1.bTargetWareHouseA := TRUE;
	_DO1.bTargetWareHouseB := FALSE;
ELSIF WareHouseSelect = E_WareHouse.WareHouseB THEN
	_DO1.bTargetWareHouseA := FALSE;
	_DO1.bTargetWareHouseB := TRUE;
ELSE
	_DO1.bTargetWareHouseA := FALSE;
	_DO1.bTargetWareHouseB := FALSE;
END_IF

// Assign coordinates 
_Layer.nInt := info.Layer;
_Slide.nInt := info.Slide;

// Send Layer data to Robot
_DO1.nLayer1 := _Layer.BitList.Bit0;
_DO1.nLayer2 := _Layer.BitList.Bit1;
_DO1.nLayer3 := _Layer.BitList.Bit2;
_DO1.nLayer4 := _Layer.BitList.Bit3;

// Send Slide data to Robot
_DO1.nSlide1 := _Slide.BitList.Bit0;
_DO1.nSlide2 := _Slide.BitList.Bit1;
_DO1.nSlide3 := _Slide.BitList.Bit2;
_DO1.nSlide4 := _Slide.BitList.Bit3;
_DO1.nSlide5 := _Slide.BitList.Bit4;

// Send action data to robot
_DO1.bGet := TRUE; // PickUp
// Send execute command 
_DO1.bExecute := TRUE;
_DO1.bContinue := BoxReady_1st;
M_StartWareHousePickUpBox_ClampA := TRUE; // Method end
END_METHOD

METHOD M_StartWareHousePickUpBox_ClampB : BOOL
VAR_INPUT
	WareHouseSelect : E_WareHouse;
	Info : ST_WareHouseCoordinates; // Input Warehouse with robot move parameter for pickup box;
	BoxReady_2nd : BOOL;
END_VAR
VAR_INST
	_Layer : ST_IntToBool;
	_Slide : ST_IntToBool;
END_VAR
// Send target warehouse to robot
IF WareHouseSelect = E_WareHouse.WareHouseA THEN
    _DO2.bTargetWareHouseA := TRUE;
    _DO2.bTargetWareHouseB := FALSE;
ELSIF WareHouseSelect = E_WareHouse.WareHouseB THEN
    _DO2.bTargetWareHouseA := FALSE;
    _DO2.bTargetWareHouseB := TRUE;
ELSE
    _DO2.bTargetWareHouseA := FALSE;
    _DO2.bTargetWareHouseB := FALSE;
END_IF

// Assign coordinates 
_Layer.nInt := info.Layer;
_Slide.nInt := info.Slide;

// Send Layer data to Robot
_DO2.nLayer1 := _Layer.BitList.Bit0;
_DO2.nLayer2 := _Layer.BitList.Bit1;
_DO2.nLayer3 := _Layer.BitList.Bit2;
_DO2.nLayer4 := _Layer.BitList.Bit3;

// Send Slide data to Robot
_DO2.nSlide1 := _Slide.BitList.Bit0;
_DO2.nSlide2 := _Slide.BitList.Bit1;
_DO2.nSlide3 := _Slide.BitList.Bit2;
_DO2.nSlide4 := _Slide.BitList.Bit3;
_DO2.nSlide5 := _Slide.BitList.Bit4;

// Send action data to robot
_DO2.bGet := TRUE; // PickUp
// Send execute command 
_DO2.bExecute := TRUE;
_DO2.bContinue:=BoxReady_2nd;
M_StartWareHousePickUpBox_ClampB := TRUE; // Method end
END_METHOD

METHOD M_StartWareHousePickUpBox_ClampBoth : BOOL
VAR_INPUT
	WareHouseSelect : E_WareHouse;
	ClampA_Info : ST_WareHouseCoordinates; // Input Warehouse with robot move parameter for pickup box;
	ClampB_Info : ST_WareHouseCoordinates; // Input Warehouse with robot move parameter for pickup box;
	BoxReady_1st : BOOL; // Box is arrived, ready to pickup
	BoxReady_2nd : BOOL; // Box is arrived, ready to pickup
END_VAR
VAR_OUTPUT
	Error : BOOL;
	ErrMsg :T_MaxString;
END_VAR
VAR_INST
	_LayerClampA : ST_IntToBool;
	_SlideClampA : ST_IntToBool;
	_LayerClampB : ST_IntToBool;
	_SlideClampB : ST_IntToBool;
END_VAR
// Set target warehouse
CASE WareHouseSelect OF
    E_WareHouse.WareHouseA:
        _DO1.bTargetWareHouseA := TRUE;
        _DO1.bTargetWareHouseB := FALSE;
        _DO2.bTargetWareHouseA := TRUE;
        _DO2.bTargetWareHouseB := FALSE;
    E_WareHouse.WareHouseB:
        _DO1.bTargetWareHouseA := FALSE;
        _DO1.bTargetWareHouseB := TRUE;
        _DO2.bTargetWareHouseA := FALSE;
        _DO2.bTargetWareHouseB := TRUE;
ELSE
    _DO1.bTargetWareHouseA := FALSE;
    _DO1.bTargetWareHouseB := FALSE;
    _DO2.bTargetWareHouseA := FALSE;
    _DO2.bTargetWareHouseB := FALSE;
    Error                  := TRUE;
    ErrMsg                 := 'Clamp target warehouse out of range';
    RETURN;
END_CASE

// Assign coordinates 
_LayerClampA.nInt := ClampA_Info.Layer;
_SlideClampA.nInt := ClampA_Info.Slide;
_LayerClampB.nInt := ClampB_Info.Layer;
_SlideClampB.nInt := ClampB_Info.Slide;

// Send Layer data to Robot
_DO1.nLayer1 := _LayerClampA.BitList.Bit0;
_DO1.nLayer2 := _LayerClampA.BitList.Bit1;
_DO1.nLayer3 := _LayerClampA.BitList.Bit2;
_DO1.nLayer4 := _LayerClampA.BitList.Bit3;

_DO2.nLayer1 := _LayerClampB.BitList.Bit0;
_DO2.nLayer2 := _LayerClampB.BitList.Bit1;
_DO2.nLayer3 := _LayerClampB.BitList.Bit2;
_DO2.nLayer4 := _LayerClampB.BitList.Bit3;
// Send Slide data to Robot
_DO1.nSlide1 := _SlideClampA.BitList.Bit0;
_DO1.nSlide2 := _SlideClampA.BitList.Bit1;
_DO1.nSlide3 := _SlideClampA.BitList.Bit2;
_DO1.nSlide4 := _SlideClampA.BitList.Bit3;
_DO1.nSlide5 := _SlideClampA.BitList.Bit4;

_DO2.nSlide1 := _SlideClampB.BitList.Bit0;
_DO2.nSlide2 := _SlideClampB.BitList.Bit1;
_DO2.nSlide3 := _SlideClampB.BitList.Bit2;
_DO2.nSlide4 := _SlideClampB.BitList.Bit3;
_DO2.nSlide5 := _SlideClampB.BitList.Bit4;

// Send action data to robot
_DO1.bGet := TRUE; // ClampA PickUp
_DO2.bGet := TRUE; // ClampB PickUp
// Send execute command 
_DO1.bExecute := NOT Error;
_DO2.bExecute := NOT Error;

_DO1.bContinue := BoxReady_1st;
_DO2.bContinue := BoxReady_2nd;

M_StartWareHousePickUpBox_ClampBoth := NOT Error; // Method end
END_METHOD

METHOD M_StartWareHousePlaceBox_ClampA : Bool
VAR_INPUT
	WareHouseSelect : E_WareHouse;
	Info : ST_WareHouseCoordinates; // Input Warehouse with robot move parameter for pickup box;
	BoxReady_1st : BOOL;
END_VAR
VAR_INST
	_Layer : ST_IntToBool;
	_Slide : ST_IntToBool;
END_VAR
// Send target warehouse to robot
IF WareHouseSelect = E_WareHouse.WareHouseA THEN
	_DO1.bTargetWareHouseA := TRUE;
	_DO1.bTargetWareHouseB := FALSE;
ELSIF WareHouseSelect = E_WareHouse.WareHouseB THEN
	_DO1.bTargetWareHouseA := FALSE;
	_DO1.bTargetWareHouseB := TRUE;
ELSE
	_DO1.bTargetWareHouseA := FALSE;
	_DO1.bTargetWareHouseB := FALSE;
END_IF

// Assign coordinates 
_Layer.nInt := info.Layer;
_Slide.nInt := info.Slide;

// Send Layer data to Robot
_DO1.nLayer1 := _Layer.BitList.Bit0;
_DO1.nLayer2 := _Layer.BitList.Bit1;
_DO1.nLayer3 := _Layer.BitList.Bit2;
_DO1.nLayer4 := _Layer.BitList.Bit3;

// Send Slide data to Robot
_DO1.nSlide1 := _Slide.BitList.Bit0;
_DO1.nSlide2 := _Slide.BitList.Bit1;
_DO1.nSlide3 := _Slide.BitList.Bit2;
_DO1.nSlide4 := _Slide.BitList.Bit3;
_DO1.nSlide5 := _Slide.BitList.Bit4;

// Send action data to robot
_DO1.bGet := FALSE; // PickUp
// Send execute command 
_DO1.bExecute := TRUE;
_DO1.bContinue := BoxReady_1st;
M_StartWareHousePlaceBox_ClampA := TRUE; // Method end
END_METHOD

METHOD M_StartWareHousePlaceBox_ClampB : BOOL
VAR_INPUT
	WareHouseSelect : E_WareHouse;
	Info : ST_WareHouseCoordinates; // Input Warehouse with robot move parameter for pickup box;
	BoxReady_2nd : BOOL;
END_VAR
VAR_INST
	_Layer : ST_IntToBool;
	_Slide : ST_IntToBool;
END_VAR
// Send target warehouse to robot
IF WareHouseSelect = E_WareHouse.WareHouseA THEN
    _DO2.bTargetWareHouseA := TRUE;
    _DO2.bTargetWareHouseB := FALSE;
ELSIF WareHouseSelect = E_WareHouse.WareHouseB THEN
    _DO2.bTargetWareHouseA := FALSE;
    _DO2.bTargetWareHouseB := TRUE;
ELSE
    _DO2.bTargetWareHouseA := FALSE;
    _DO2.bTargetWareHouseB := FALSE;
END_IF

// Assign coordinates 
_Layer.nInt := info.Layer;
_Slide.nInt := info.Slide;

// Send Layer data to Robot
_DO2.nLayer1 := _Layer.BitList.Bit0;
_DO2.nLayer2 := _Layer.BitList.Bit1;
_DO2.nLayer3 := _Layer.BitList.Bit2;
_DO2.nLayer4 := _Layer.BitList.Bit3;

// Send Slide data to Robot
_DO2.nSlide1 := _Slide.BitList.Bit0;
_DO2.nSlide2 := _Slide.BitList.Bit1;
_DO2.nSlide3 := _Slide.BitList.Bit2;
_DO2.nSlide4 := _Slide.BitList.Bit3;
_DO2.nSlide5 := _Slide.BitList.Bit4;

// Send action data to robot
_DO2.bGet := FALSE; // PickUp
// Send execute command 
_DO2.bExecute := TRUE;
_DO2.bContinue:=BoxReady_2nd;
M_StartWareHousePlaceBox_ClampB := TRUE; // Method end
END_METHOD

METHOD M_StartWareHousePlaceUpBox_ClampBoth : BOOL
VAR_INPUT
	WareHouseSelect : E_WareHouse;
	ClampA_Info : ST_WareHouseCoordinates; // Input Warehouse with robot move parameter for pickup box;
	ClampB_Info : ST_WareHouseCoordinates; // Input Warehouse with robot move parameter for pickup box;
	BoxReady_1st : BOOL; // Box is arrived, ready to pickup
	BoxReady_2nd : BOOL; // Box is arrived, ready to pickup
END_VAR
VAR_OUTPUT
	Error : BOOL;
	ErrMsg :T_MaxString;
END_VAR
VAR_INST
	_LayerClampA : ST_IntToBool;
	_SlideClampA : ST_IntToBool;
	_LayerClampB : ST_IntToBool;
	_SlideClampB : ST_IntToBool;
END_VAR
// Set target warehouse
CASE WareHouseSelect OF
    E_WareHouse.WareHouseA:
        _DO1.bTargetWareHouseA := TRUE;
        _DO1.bTargetWareHouseB := FALSE;
        _DO2.bTargetWareHouseA := TRUE;
        _DO2.bTargetWareHouseB := FALSE;
    E_WareHouse.WareHouseB:
        _DO1.bTargetWareHouseA := FALSE;
        _DO1.bTargetWareHouseB := TRUE;
        _DO2.bTargetWareHouseA := FALSE;
        _DO2.bTargetWareHouseB := TRUE;
ELSE
    _DO1.bTargetWareHouseA := FALSE;
    _DO1.bTargetWareHouseB := FALSE;
    _DO2.bTargetWareHouseA := FALSE;
    _DO2.bTargetWareHouseB := FALSE;
    Error                  := TRUE;
    ErrMsg                 := 'Clamp target warehouse out of range';
    RETURN;
END_CASE

// Assign coordinates 
_LayerClampA.nInt := ClampA_Info.Layer;
_SlideClampA.nInt := ClampA_Info.Slide;
_LayerClampB.nInt := ClampB_Info.Layer;
_SlideClampB.nInt := ClampB_Info.Slide;

// Send Layer data to Robot
_DO1.nLayer1 := _LayerClampA.BitList.Bit0;
_DO1.nLayer2 := _LayerClampA.BitList.Bit1;
_DO1.nLayer3 := _LayerClampA.BitList.Bit2;
_DO1.nLayer4 := _LayerClampA.BitList.Bit3;

_DO2.nLayer1 := _LayerClampB.BitList.Bit0;
_DO2.nLayer2 := _LayerClampB.BitList.Bit1;
_DO2.nLayer3 := _LayerClampB.BitList.Bit2;
_DO2.nLayer4 := _LayerClampB.BitList.Bit3;
// Send Slide data to Robot
_DO1.nSlide1 := _SlideClampA.BitList.Bit0;
_DO1.nSlide2 := _SlideClampA.BitList.Bit1;
_DO1.nSlide3 := _SlideClampA.BitList.Bit2;
_DO1.nSlide4 := _SlideClampA.BitList.Bit3;
_DO1.nSlide5 := _SlideClampA.BitList.Bit4;

_DO2.nSlide1 := _SlideClampB.BitList.Bit0;
_DO2.nSlide2 := _SlideClampB.BitList.Bit1;
_DO2.nSlide3 := _SlideClampB.BitList.Bit2;
_DO2.nSlide4 := _SlideClampB.BitList.Bit3;
_DO2.nSlide5 := _SlideClampB.BitList.Bit4;

// Send action data to robot
_DO1.bGet := FALSE; // ClampA PickUp
_DO2.bGet := FALSE; // ClampB PickUp
// Send execute command 
_DO1.bExecute := NOT Error;
_DO2.bExecute := NOT Error;

_DO1.bContinue := BoxReady_1st;
_DO2.bContinue := BoxReady_2nd;

M_StartWareHousePlaceUpBox_ClampBoth := NOT Error; // Method end
END_METHOD

METHOD M_SwitchRSR3 : BOOL
VAR_INPUT
END_VAR
END_METHOD

PROPERTY Read_OffsetP : INT
GET
Read_OffsetP := _DI6;
END_GET
END_PROPERTY

PROPERTY Read_OffsetR : INT
GET
Read_OffsetR := _DI7;
END_GET
END_PROPERTY

PROPERTY Read_OffsetW : INT
GET
Read_OffsetW := _DI5;
END_GET
END_PROPERTY

PROPERTY Read_OffsetX : INT
GET
Read_OffsetX := _DI2;
END_GET
END_PROPERTY

PROPERTY Read_OffsetY : INT
GET
Read_OffsetY := _DI3;
END_GET
END_PROPERTY

PROPERTY Read_OffsetZ : INT
GET
Read_OffsetZ := _DI4;
END_GET
END_PROPERTY

PROPERTY ReadDataCommand : BOOL;
SET
_DO6.ReadPara_Execute := BOOL_TO_BIT(ReadDataCommand);
END_SET
END_PROPERTY

PROPERTY ReadWrite_Address : Int
SET
_Do14 := ReadWrite_Address;
END_SET
END_PROPERTY

PROPERTY ReadWrite_Area : E_RobotArea
SET
_Do13 := ReadWrite_Area;
END_SET
END_PROPERTY

(* This variable is used to define read/write offset data clamp A
*)
PROPERTY ReadWrite_ClampA : BOOL
SET
_DO6.ClampA :=  BOOL_TO_BIT(ReadWrite_ClampA );
END_SET
END_PROPERTY

(* This variable is used to define read/write offset data clamp B
*)
PROPERTY ReadWrite_ClampB : BOOL
SET
_DO6.ClampB :=BOOL_TO_BIT( ReadWrite_ClampB);
END_SET
END_PROPERTY

(* This variable is used to define read/write offset data warehouse A
*)
PROPERTY ReadWrite_WareHouseA : BOOL
SET
_DO6.WareHouseA := BOOL_TO_BIT(ReadWrite_WareHouseA);
END_SET
END_PROPERTY

(* This variable is used to define read/write offset data warehouse B
*)
PROPERTY ReadWrite_WareHouseB : BOOL
SET
_DO6.WarehouseB := BOOL_TO_BIT(ReadWrite_WareHouseB);
END_SET
END_PROPERTY

(*Fanuc robot ready to work for command (Warehouse、AbsMove)*)
PROPERTY ReadyOperation : Bool
GET
ReadyOperation := _RSR1_Ready;
END_GET
END_PROPERTY

PROPERTY ReadySetParameter : Bool
GET
ReadySetParameter := _RSR3_Ready;
END_GET
END_PROPERTY

METHOD ReBoot
VAR_INPUT
END_VAR
eState := E_MethodStatus_Basic.STATE_DORMANT;
END_METHOD

PROPERTY SlideIndex : INT
SET
_DO16 := SlideIndex;
END_SET
END_PROPERTY

PROPERTY Status : ST_FanucUI1
GET
Status := _UI1;
END_GET
END_PROPERTY

METHOD Update : BOOL
VAR_INPUT
END_VAR
// Robot -> PLC 4 byte 外圍設備Output(Fanuc Robot的外圍)
MEMMOVE(
destAddr:=ADR(_UO1)
,srcAddr:=ADR(_rawIn_UI[0])
,n:=4
);

